KUKA KRL program: MyProgram_223().src

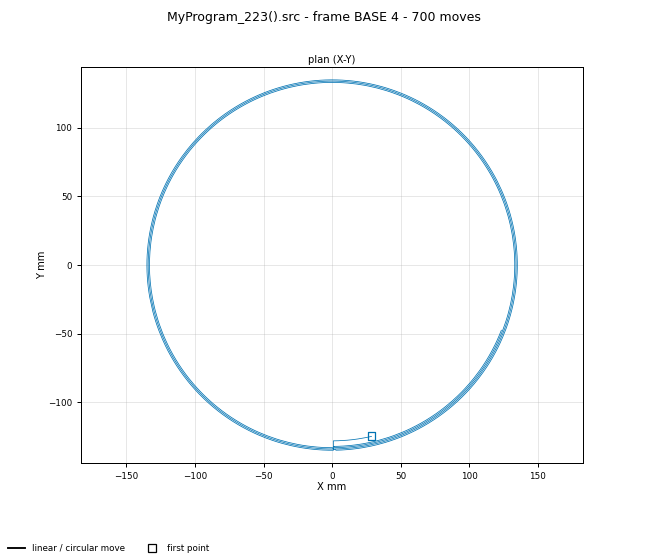
[picture p0: tool path of MyProgram_223().src in frame BASE 4, 700 of 700 moves have a stored position in this frame; points joined in program order, loops and branches not executed]
&ACCESS RVP
&REL 1
&PARAM TEMPLATE = C:\KRC\Roboter\Template\vorgabe
&PARAM EDITMASK = *
DEF MyProgram_223()
; ---- Setting reference (Base) ----
$BASE = BASE_DATA[4]

; --------------------------
; ---- Setting tool (TCP) ----
$TOOL = TOOL_DATA[3]
; --------------------------

$VEL.CP = VEL_APROX_PRINT
Startdeposition()
$VEL.CP = VEL_PRINT
LIN {X 28.7069,Y -124.9653,Z 154,A -77.9995,B 16.837,C -0.17,E1 16.8732,E2 526.8785} C_DIS
LIN {X 25.0095,Y -125.7587,Z 154,A -79.6825,B 16.837,C -0.1689,E1 16.8686,E2 528.562} C_DIS
LIN {X 21.848,Y -126.3473,Z 154,A -81.1205,B 16.837,C -0.1678,E1 16.8647,E2 530.0012} C_DIS
LIN {X 18.7921,Y -126.8373,Z 154,A -82.6165,B 16.837,C -0.1631,E1 16.8605,E2 531.5113} C_DIS
LIN {X 14.8187,Y -127.3616,Z 154,A -84.2756,B 16.837,C -0.1666,E1 16.8559,E2 533.1562} C_DIS
LIN {X 10.9976,Y -127.7479,Z 154,A -86.0056,B 16.837,C -0.1654,E1 16.8511,E2 534.8888} C_DIS
LIN {X 7.8618,Y -127.979,Z 154,A -87.4025,B 16.837,C -0.1651,E1 16.8472,E2 536.2856} C_DIS
LIN {X 4.7214,Y -128.1337,Z 154,A -88.9391,B 16.837,C -0.1603,E1 16.8429,E2 537.8382} C_DIS
LIN {X 0.8945,Y -128.2158,Z 154,A -89.9476,B 16.8368,C -0.1836,E1 16.8403,E2 538.7658} C_DIS
Enddeposition()
LIN {X 0.956,Y -135.0652,Z 155,A -92.2776,B 24.9684,C -1.2991,E1 25.0025,E2 538.84} C_DIS
Startdeposition()
$VEL.CP = VEL_PRINT
LIN {X -2.5758,Y -135.0444,Z 155,A -94.5411,B 24.9704,C -1.2578,E1 24.996,E2 541.2013} C_DIS
LIN {X -6.7331,Y -134.9006,Z 155,A -96.2372,B 24.9702,C -1.2612,E1 24.9912,E2 542.8895} C_DIS
LIN {X -10.9178,Y -134.6272,Z 155,A -98.0533,B 24.9703,C -1.2593,E1 24.9862,E2 544.711} C_DIS
LIN {X -14.6224,Y -134.2747,Z 155,A -99.5996,B 24.9703,C -1.2612,E1 24.9819,E2 546.2538} C_DIS
LIN {X -18.9041,Y -133.7391,Z 155,A -101.4287,B 24.9702,C -1.2616,E1 24.9768,E2 548.0831} C_DIS
LIN {X -22.4797,Y -133.1848,Z 155,A -102.9613,B 24.9702,C -1.2622,E1 24.9726,E2 549.6158} C_DIS
LIN {X -26.677,Y -132.4079,Z 155,A -104.759,B 24.9701,C -1.2636,E1 24.9677,E2 551.4121} C_DIS
LIN {X -30.089,Y -131.6741,Z 155,A -106.2282,B 24.9701,C -1.2649,E1 24.9637,E2 552.8801} C_DIS
LIN {X -33.3739,Y -130.8802,Z 155,A -107.6389,B 24.9699,C -1.2669,E1 24.9599,E2 554.2879} C_DIS
LIN {X -36.516,Y -130.0385,Z 155,A -109.0601,B 24.9699,C -1.2657,E1 24.956,E2 555.7143} C_DIS
LIN {X -39.7548,Y -129.0853,Z 155,A -110.482,B 24.9699,C -1.2672,E1 24.9522,E2 557.1349} C_DIS
LIN {X -43.4103,Y -127.9044,Z 155,A -112.2658,B 24.9702,C -1.2605,E1 24.9474,E2 558.9378} C_DIS
LIN {X -48.0128,Y -126.2483,Z 155,A -114.1681,B 24.9697,C -1.2714,E1 24.9425,E2 560.8182} C_DIS
LIN {X -50.9174,Y -125.104,Z 155,A -115.4973,B 24.9697,C -1.2725,E1 24.9391,E2 562.1477} C_DIS
LIN {X -53.8737,Y -123.8591,Z 155,A -116.8849,B 24.9697,C -1.2726,E1 24.9355,E2 563.5383} C_DIS
LIN {X -57.0265,Y -122.4397,Z 155,A -118.3499,B 24.9696,C -1.2744,E1 24.9318,E2 565.0027} C_DIS
LIN {X -60.55,Y -120.7382,Z 155,A -120.1373,B 24.9698,C -1.2699,E1 24.9273,E2 566.8054} C_DIS
LIN {X -64.3446,Y -118.7594,Z 155,A -121.9404,B 24.9696,C -1.273,E1 24.9228,E2 568.6063} C_DIS
LIN {X -68.1625,Y -116.6098,Z 155,A -123.8138,B 24.9696,C -1.2749,E1 24.9183,E2 570.4805} C_DIS
LIN {X -72.0026,Y -114.2783,Z 155,A -125.7043,B 24.9694,C -1.2787,E1 24.9138,E2 572.3682} C_DIS
LIN {X -75.5548,Y -111.9616,Z 155,A -127.5227,B 24.9693,C -1.2806,E1 24.9096,E2 574.1878} C_DIS
LIN {X -79.2894,Y -109.3484,Z 155,A -129.4475,B 24.9691,C -1.2844,E1 24.9052,E2 576.1102} C_DIS
LIN {X -82.9569,Y -106.5932,Z 155,A -131.4123,B 24.969,C -1.287,E1 24.9008,E2 578.076} C_DIS
LIN {X -86.4643,Y -103.7689,Z 155,A -133.3577,B 24.9689,C -1.2889,E1 24.8966,E2 580.0244} C_DIS
LIN {X -89.8678,Y -100.8354,Z 155,A -135.2713,B 24.9687,C -1.2924,E1 24.8926,E2 581.9372} C_DIS
LIN {X -93.2442,Y -97.7211,Z 155,A -137.1683,B 24.9684,C -1.2991,E1 24.8887,E2 583.826} C_DIS
LIN {X -96.9915,Y -94.0028,Z 155,A -139.3932,B 24.9681,C -1.3047,E1 24.8844,E2 586.047} C_DIS
LIN {X -99.861,Y -90.9491,Z 155,A -141.2062,B 24.9681,C -1.3069,E1 24.8809,E2 587.8626} C_DIS
LIN {X -102.662,Y -87.7755,Z 155,A -142.9452,B 24.9677,C -1.314,E1 24.8778,E2 589.5927} C_DIS
LIN {X -105.1,Y -84.8403,Z 155,A -144.6551,B 24.9677,C -1.3133,E1 24.8747,E2 591.3121} C_DIS
LIN {X -108.2093,Y -80.8373,Z 155,A -146.8037,B 24.9674,C -1.3188,E1 24.8711,E2 593.458} C_DIS
LIN {X -110.7077,Y -77.3807,Z 155,A -148.6369,B 24.9673,C -1.3222,E1 24.8681,E2 595.292} C_DIS
LIN {X -113.1135,Y -73.8196,Z 155,A -150.4801,B 24.9671,C -1.326,E1 24.8653,E2 597.1353} C_DIS
LIN {X -115.3987,Y -70.1936,Z 155,A -152.3394,B 24.9669,C -1.3289,E1 24.8625,E2 598.9974} C_DIS
LIN {X -117.7263,Y -66.2149,Z 155,A -154.2561,B 24.9666,C -1.3362,E1 24.8599,E2 600.9066} C_DIS
LIN {X -119.7417,Y -62.4932,Z 155,A -155.9961,B 24.9662,C -1.344,E1 24.8576,E2 602.6371} C_DIS
LIN {X -121.6486,Y -58.6962,Z 155,A -157.6914,B 24.9656,C -1.3545,E1 24.8555,E2 604.3166} C_DIS
LIN {X -123.7406,Y -54.1479,Z 155,A -159.8366,B 24.9654,C -1.3596,E1 24.853,E2 606.4614} C_DIS
LIN {X -125.3816,Y -50.2287,Z 155,A -161.6964,B 24.9652,C -1.3621,E1 24.851,E2 608.3256} C_DIS
LIN {X -126.4676,Y -47.427,Z 155,A -163.026,B 24.9652,C -1.3633,E1 24.8497,E2 609.66} C_DIS
LIN {X -127.6173,Y -44.2406,Z 155,A -164.4544,B 24.9649,C -1.3681,E1 24.8484,E2 611.085} C_DIS
LIN {X -128.7101,Y -40.953,Z 155,A -165.9753,B 24.9649,C -1.3701,E1 24.8471,E2 612.6098} C_DIS
LIN {X -129.859,Y -37.1578,Z 155,A -167.9428,B 24.9653,C -1.3613,E1 24.8455,E2 614.6097} C_DIS
LIN {X -130.7137,Y -34.0292,Z 155,A -169.0198,B 24.9643,C -1.3802,E1 24.8448,E2 615.6478} C_DIS
LIN {X -133.0003,Y -23.5463,Z 155,A -173.6124,B 24.9637,C -1.3927,E1 24.8421,E2 620.2378} C_DIS
LIN {X -133.6072,Y -19.827,Z 155,A -175.3609,B 24.9637,C -1.3905,E1 24.8413,E2 622.002} C_DIS
LIN {X -134.12,Y -15.9779,Z 155,A -176.8994,B 24.9632,C -1.4012,E1 24.8408,E2 623.5241} C_DIS
LIN {X -134.4898,Y -12.4963,Z 155,A -178.3737,B 24.9629,C -1.4066,E1 24.8404,E2 624.9944} C_DIS
LIN {X -134.7979,Y -8.5494,Z 155,A 179.9081,B 24.9627,C -1.4102,E1 24.84,E2 626.7143} C_DIS
LIN {X -134.9759,Y -5.0083,Z 155,A 178.3069,B 24.9627,C -1.4104,E1 24.8399,E2 628.3247} C_DIS
LIN {X -135.0684,Y -0.5524,Z 155,A 176.4249,B 24.9624,C -1.4171,E1 24.8398,E2 630.2022} C_DIS
LIN {X -135.0185,Y 3.6788,Z 155,A 174.6963,B 24.9619,C -1.4263,E1 24.8398,E2 631.9192} C_DIS
LIN {X -134.8642,Y 7.4574,Z 155,A 172.9572,B 24.9619,C -1.425,E1 24.8401,E2 633.6718} C_DIS
LIN {X -134.5797,Y 11.4806,Z 155,A 171.3594,B 24.9614,C -1.4362,E1 24.8405,E2 635.2525} C_DIS
LIN {X -134.165,Y 15.6009,Z 155,A 169.5519,B 24.9612,C -1.4395,E1 24.841,E2 637.0629} C_DIS
LIN {X -133.7051,Y 19.1415,Z 155,A 168.0667,B 24.9608,C -1.446,E1 24.8416,E2 638.5416} C_DIS
LIN {X -133.0954,Y 23.0147,Z 155,A 166.2283,B 24.961,C -1.4429,E1 24.8424,E2 640.3984} C_DIS
LIN {X -132.3123,Y 27.1467,Z 155,A 164.5508,B 24.9604,C -1.454,E1 24.8433,E2 642.0594} C_DIS
LIN {X -131.1469,Y 32.3169,Z 155,A 162.3649,B 24.9598,C -1.4643,E1 24.8447,E2 644.2333} C_DIS
LIN {X -130.3875,Y 35.2526,Z 155,A 160.9043,B 24.9601,C -1.46,E1 24.8457,E2 645.7127} C_DIS
LIN {X -129.1991,Y 39.3831,Z 155,A 158.5311,B 24.9612,C -1.4393,E1 24.8477,E2 648.1491} C_DIS
LIN {X -127.5792,Y 44.3504,Z 155,A 156.9773,B 24.959,C -1.4785,E1 24.849,E2 649.6183} C_DIS
LIN {X -126.4051,Y 47.5939,Z 155,A 155.4977,B 24.9588,C -1.4823,E1 24.8504,E2 651.0971} C_DIS
LIN {X -125.2195,Y 50.6307,Z 155,A 154.1008,B 24.9586,C -1.486,E1 24.8519,E2 652.493} C_DIS
LIN {X -123.8761,Y 53.8345,Z 155,A 152.6264,B 24.9584,C -1.4906,E1 24.8535,E2 653.9647} C_DIS
LIN {X -122.507,Y 56.8809,Z 155,A 151.1945,B 24.9582,C -1.4942,E1 24.8552,E2 655.3957} C_DIS
LIN {X -120.9936,Y 60.0334,Z 155,A 149.6811,B 24.958,C -1.4973,E1 24.857,E2 656.9101} C_DIS
LIN {X -119.2067,Y 63.5116,Z 155,A 147.8717,B 24.9581,C -1.4949,E1 24.8594,E2 658.7348} C_DIS
LIN {X -116.8772,Y 67.7024,Z 155,A 145.8996,B 24.9576,C -1.504,E1 24.8621,E2 660.6955} C_DIS
LIN {X -114.4989,Y 71.6521,Z 155,A 143.9181,B 24.9574,C -1.5084,E1 24.865,E2 662.6766} C_DIS
LIN {X -112.0741,Y 75.3886,Z 155,A 141.9947,B 24.9572,C -1.5122,E1 24.8679,E2 664.6007} C_DIS
LIN {X -109.5159,Y 79.0583,Z 155,A 140.1208,B 24.9568,C -1.5187,E1 24.8709,E2 666.4682} C_DIS
LIN {X -105.4703,Y 84.3802,Z 155,A 137.3252,B 24.9562,C -1.5284,E1 24.8757,E2 669.254} C_DIS
LIN {X -101.5038,Y 89.1125,Z 155,A 134.5151,B 24.9564,C -1.526,E1 24.8808,E2 672.0828} C_DIS
LIN {X -97.5119,Y 93.4631,Z 155,A 132.2969,B 24.9552,C -1.5465,E1 24.885,E2 674.2618} C_DIS
LIN {X -95.259,Y 95.7581,Z 155,A 130.7619,B 24.9555,C -1.5415,E1 24.888,E2 675.8154} C_DIS
LIN {X -92.1865,Y 98.7196,Z 155,A 128.877,B 24.9555,C -1.5421,E1 24.8919,E2 677.7064} C_DIS
LIN {X -88.0432,Y 102.4319,Z 155,A 126.8279,B 24.9542,C -1.5631,E1 24.8961,E2 679.7137} C_DIS
LIN {X -85.7976,Y 104.3208,Z 155,A 125.2543,B 24.955,C -1.5495,E1 24.8995,E2 681.3255} C_DIS
LIN {X -82.2968,Y 107.1038,Z 155,A 122.8357,B 24.9563,C -1.5279,E1 24.905,E2 683.8044} C_DIS
LIN {X -78.1726,Y 110.1502,Z 155,A 121.4737,B 24.9537,C -1.5728,E1 24.9079,E2 685.0644} C_DIS
LIN {X -73.9894,Y 113.0026,Z 155,A 119.0337,B 24.9543,C -1.5625,E1 24.9136,E2 687.537} C_DIS
LIN {X -70.0577,Y 115.4809,Z 155,A 117.0561,B 24.9541,C -1.566,E1 24.9183,E2 689.5126} C_DIS
LIN {X -66.2162,Y 117.7256,Z 155,A 115.1687,B 24.9539,C -1.5694,E1 24.9228,E2 691.3975} C_DIS
LIN {X -62.6191,Y 119.6756,Z 155,A 113.5082,B 24.9534,C -1.5762,E1 24.9269,E2 693.0464} C_DIS
LIN {X -59.6022,Y 121.2063,Z 155,A 112.069,B 24.9534,C -1.5784,E1 24.9305,E2 694.4842} C_DIS
LIN {X -56.3004,Y 122.7755,Z 155,A 110.5474,B 24.9531,C -1.5823,E1 24.9343,E2 696.0005} C_DIS
LIN {X -53.2438,Y 124.1315,Z 155,A 109.0926,B 24.9531,C -1.5826,E1 24.938,E2 697.458} C_DIS
LIN {X -49.3123,Y 125.7451,Z 155,A 107.2368,B 24.9531,C -1.5825,E1 24.9429,E2 699.3181} C_DIS
LIN {X -45.9259,Y 127.0206,Z 155,A 105.74,B 24.9528,C -1.5864,E1 24.9468,E2 700.8085} C_DIS
LIN {X -42.4672,Y 128.2185,Z 155,A 104.2256,B 24.9526,C -1.5903,E1 24.9507,E2 702.3166} C_DIS
LIN {X -39.232,Y 129.2453,Z 155,A 102.7595,B 24.9526,C -1.5907,E1 24.9547,E2 703.7844} C_DIS
LIN {X -35.3424,Y 130.3635,Z 155,A 100.9587,B 24.9527,C -1.5882,E1 24.9595,E2 705.5939} C_DIS
LIN {X -31.7612,Y 131.2809,Z 155,A 99.444,B 24.9525,C -1.5925,E1 24.9636,E2 707.1005} C_DIS
LIN {X -28.1853,Y 132.0951,Z 155,A 97.9093,B 24.9523,C -1.595,E1 24.9678,E2 708.6312} C_DIS
LIN {X -24.1975,Y 132.8838,Z 155,A 96.1246,B 24.9524,C -1.5933,E1 24.9727,E2 710.4219} C_DIS
LIN {X -20.4636,Y 133.5093,Z 155,A 94.597,B 24.9521,C -1.5985,E1 24.9769,E2 711.9386} C_DIS
LIN {X -17.178,Y 133.9721,Z 155,A 93.0679,B 24.9524,C -1.5931,E1 24.9811,E2 713.4815} C_DIS
LIN {X -12.8968,Y 134.4513,Z 155,A 91.3198,B 24.9521,C -1.5982,E1 24.986,E2 715.2187} C_DIS
LIN {X -8.8291,Y 134.7806,Z 155,A 89.5073,B 24.9523,C -1.5948,E1 24.991,E2 717.04} C_DIS
LIN {X -4.9442,Y 134.9784,Z 155,A 87.8488,B 24.9523,C -1.5948,E1 24.9957,E2 718.6986} C_DIS
LIN {X -0.6766,Y 135.0669,Z 155,A 86.1042,B 24.9521,C -1.5988,E1 25.0005,E2 720.4341} C_DIS
LIN {X 3.559,Y 135.0218,Z 155,A 84.3207,B 24.9521,C -1.5997,E1 25.0055,E2 722.2151} C_DIS
LIN {X 7.3645,Y 134.8688,Z 155,A 82.605,B 24.9524,C -1.5945,E1 25.0103,E2 723.9426} C_DIS
LIN {X 11.3614,Y 134.5898,Z 155,A 81.0168,B 24.952,C -1.6003,E1 25.0147,E2 725.5163} C_DIS
LIN {X 15.2359,Y 134.2085,Z 155,A 79.2316,B 24.9525,C -1.593,E1 25.0197,E2 727.3176} C_DIS
LIN {X 19.1015,Y 133.7109,Z 155,A 77.7249,B 24.952,C -1.6003,E1 25.0238,E2 728.8057} C_DIS
LIN {X 22.5739,Y 133.169,Z 155,A 76.1081,B 24.9524,C -1.5932,E1 25.0283,E2 730.4378} C_DIS
LIN {X 26.8961,Y 132.3633,Z 155,A 74.3688,B 24.9521,C -1.599,E1 25.033,E2 732.1613} C_DIS
LIN {X 30.2156,Y 131.6452,Z 155,A 72.9373,B 24.9521,C -1.5987,E1 25.0369,E2 733.5915} C_DIS
LIN {X 33.4163,Y 130.8694,Z 155,A 71.524,B 24.9522,C -1.597,E1 25.0408,E2 735.0067} C_DIS
LIN {X 36.6251,Y 130.008,Z 155,A 70.1141,B 24.9522,C -1.596,E1 25.0446,E2 736.4168} C_DIS
LIN {X 40.4048,Y 128.8852,Z 155,A 68.3482,B 24.9526,C -1.5897,E1 25.0493,E2 738.1943} C_DIS
LIN {X 45.0769,Y 127.3266,Z 155,A 66.3968,B 24.9523,C -1.5952,E1 25.0544,E2 740.1289} C_DIS
LIN {X 47.6833,Y 126.3716,Z 155,A 65.2107,B 24.9524,C -1.5936,E1 25.0575,E2 741.3163} C_DIS
LIN {X 50.746,Y 125.1731,Z 155,A 63.7899,B 24.9526,C -1.5908,E1 25.0612,E2 742.7406} C_DIS
LIN {X 53.8201,Y 123.8823,Z 155,A 62.393,B 24.9526,C -1.5902,E1 25.0648,E2 744.1356} C_DIS
LIN {X 56.9496,Y 122.4753,Z 155,A 60.9484,B 24.9526,C -1.589,E1 25.0685,E2 745.5794} C_DIS
LIN {X 60.0444,Y 120.9882,Z 155,A 59.4823,B 24.9528,C -1.5866,E1 25.0722,E2 747.0472} C_DIS
LIN {X 63.2089,Y 119.3659,Z 155,A 57.9622,B 24.953,C -1.584,E1 25.0759,E2 748.5694} C_DIS
LIN {X 66.9392,Y 117.316,Z 155,A 56.0485,B 24.9535,C -1.5755,E1 25.0806,E2 750.4973} C_DIS
LIN {X 70.8345,Y 115.0062,Z 155,A 54.2606,B 24.9532,C -1.5797,E1 25.0849,E2 752.2697} C_DIS
LIN {X 74.1026,Y 112.928,Z 155,A 52.5215,B 24.9537,C -1.5719,E1 25.089,E2 754.0218} C_DIS
LIN {X 77.8951,Y 110.346,Z 155,A 50.6151,B 24.9537,C -1.5707,E1 25.0933,E2 755.9245} C_DIS
LIN {X 81.529,Y 107.6892,Z 155,A 48.716,B 24.9539,C -1.5678,E1 25.0976,E2 757.8237} C_DIS
LIN {X 85.0807,Y 104.9061,Z 155,A 46.8107,B 24.9541,C -1.5646,E1 25.1018,E2 759.7293} C_DIS
LIN {X 88.2784,Y 102.2293,Z 155,A 45.0412,B 24.9543,C -1.561,E1 25.1055,E2 761.5003} C_DIS
LIN {X 91.5574,Y 99.3034,Z 155,A 43.1894,B 24.9545,C -1.5579,E1 25.1094,E2 763.3521} C_DIS
LIN {X 94.7667,Y 96.2456,Z 155,A 41.2984,B 24.9548,C -1.5532,E1 25.1132,E2 765.2462} C_DIS
LIN {X 97.9192,Y 93.0369,Z 155,A 39.433,B 24.9549,C -1.5513,E1 25.1168,E2 767.1082} C_DIS
LIN {X 100.8417,Y 89.8607,Z 155,A 37.6085,B 24.9551,C -1.5474,E1 25.1202,E2 768.9338} C_DIS
LIN {X 103.6576,Y 86.5972,Z 155,A 35.7454,B 24.9555,C -1.5411,E1 25.1236,E2 770.8032} C_DIS
LIN {X 106.466,Y 83.1206,Z 155,A 33.8428,B 24.9558,C -1.536,E1 25.1269,E2 772.7088} C_DIS
LIN {X 109.1862,Y 79.5132,Z 155,A 31.9399,B 24.956,C -1.5319,E1 25.1301,E2 774.6123} C_DIS
LIN {X 111.7145,Y 75.9199,Z 155,A 30.089,B 24.9563,C -1.5278,E1 25.133,E2 776.4639} C_DIS
LIN {X 114.2202,Y 72.0947,Z 155,A 28.1796,B 24.9565,C -1.5243,E1 25.1359,E2 778.372} C_DIS
LIN {X 116.5986,Y 68.1817,Z 155,A 26.2431,B 24.9568,C -1.5193,E1 25.1387,E2 780.3104} C_DIS
LIN {X 118.7941,Y 64.2807,Z 155,A 24.3469,B 24.9571,C -1.5141,E1 25.1412,E2 782.2089} C_DIS
LIN {X 120.525,Y 60.9688,Z 155,A 22.9027,B 24.9569,C -1.5174,E1 25.1431,E2 783.6375} C_DIS
LIN {X 121.9558,Y 58.0532,Z 155,A 21.5126,B 24.9571,C -1.5128,E1 25.1447,E2 785.0312} C_DIS
LIN {X 123.3484,Y 55.0323,Z 155,A 20.1045,B 24.9574,C -1.5088,E1 25.1464,E2 786.4411} C_DIS
LIN {X 124.7016,Y 51.8933,Z 155,A 18.6636,B 24.9576,C -1.505,E1 25.1479,E2 787.8829} C_DIS
LIN {X 125.9888,Y 48.6856,Z 155,A 17.2055,B 24.9578,C -1.501,E1 25.1494,E2 789.3423} C_DIS
LIN {X 127.4202,Y 44.809,Z 155,A 15.3011,B 24.9586,C -1.4872,E1 25.1513,E2 791.2685} C_DIS
LIN {X 128.9009,Y 40.3554,Z 155,A 13.139,B 24.9594,C -1.4715,E1 25.1531,E2 793.4554} C_DIS
LIN {X 129.9101,Y 36.9751,Z 155,A 12.0923,B 24.9583,C -1.492,E1 25.1539,E2 794.448} C_DIS
LIN {X 130.9776,Y 32.99,Z 155,A 10.2421,B 24.9589,C -1.4808,E1 25.1552,E2 796.3137} C_DIS
LIN {X 131.967,Y 28.7787,Z 155,A 8.4174,B 24.9592,C -1.4756,E1 25.1564,E2 798.1402} C_DIS
LIN {X 132.6716,Y 25.3314,Z 155,A 6.9657,B 24.9593,C -1.4731,E1 25.1571,E2 799.5894} C_DIS
LIN {X 133.2979,Y 21.8018,Z 155,A 5.4671,B 24.9596,C -1.4694,E1 25.1578,E2 801.0878} C_DIS
LIN {X 133.865,Y 17.9954,Z 155,A 3.7685,B 24.96,C -1.4604,E1 25.1585,E2 802.7978} C_DIS
LIN {X 134.3238,Y 14.1661,Z 155,A 2.1058,B 24.9604,C -1.4535,E1 25.159,E2 804.4667} C_DIS
LIN {X 134.7085,Y 9.854,Z 155,A 0.3864,B 24.9604,C -1.4541,E1 25.1594,E2 806.1746} C_DIS
LIN {X 134.9165,Y 6.416,Z 155,A -1.1834,B 24.961,C -1.4431,E1 25.1597,E2 807.7609} C_DIS
LIN {X 135.0499,Y 2.2472,Z 155,A -2.8475,B 24.961,C -1.4431,E1 25.1597,E2 809.415} C_DIS
LIN {X 135.0526,Y -2.0829,Z 155,A -4.687,B 24.9613,C -1.4369,E1 25.1597,E2 811.2582} C_DIS
LIN {X 134.9392,Y -5.9477,Z 155,A -6.3919,B 24.9618,C -1.4278,E1 25.1596,E2 812.9744} C_DIS
LIN {X 134.7122,Y -9.8033,Z 155,A -7.8928,B 24.9617,C -1.4301,E1 25.1593,E2 814.461} C_DIS
LIN {X 134.4232,Y -13.1893,Z 155,A -9.4289,B 24.9622,C -1.42,E1 25.1589,E2 816.0118} C_DIS
LIN {X 133.938,Y -17.4382,Z 155,A -11.1522,B 24.9622,C -1.4191,E1 25.1583,E2 817.7271} C_DIS
LIN {X 133.4162,Y -21.0649,Z 155,A -12.7866,B 24.9628,C -1.4094,E1 25.1576,E2 819.3746} C_DIS
LIN {X 132.6927,Y -25.2211,Z 155,A -14.4859,B 24.9628,C -1.4086,E1 25.1568,E2 821.066} C_DIS
LIN {X 131.9741,Y -28.7461,Z 155,A -15.967,B 24.963,C -1.4061,E1 25.1559,E2 822.5443} C_DIS
LIN {X 131.1265,Y -32.4017,Z 155,A -17.6861,B 24.9636,C -1.3937,E1 25.1548,E2 824.2827} C_DIS
LIN {X 130.1075,Y -36.2695,Z 155,A -19.2728,B 24.9636,C -1.3944,E1 25.1537,E2 825.8587} C_DIS
LIN {X 129.1637,Y -39.4988,Z 155,A -20.6741,B 24.9637,C -1.3912,E1 25.1525,E2 827.2594} C_DIS
LIN {X 128.1047,Y -42.8088,Z 155,A -22.1386,B 24.964,C -1.387,E1 25.1513,E2 828.7256} C_DIS
LIN {X 126.7849,Y -46.5796,Z 155,A -24.1151,B 24.9651,C -1.3658,E1 25.1494,E2 830.741} C_DIS
LIN {X 125.5935,Y -49.7023,Z 155,A -25.2102,B 24.9644,C -1.3794,E1 25.1483,E2 831.798} C_DIS
LIN {X 124.5325,Y -52.2983,Z 155,A -26.5775,B 24.9651,C -1.3657,E1 25.1468,E2 833.1901} C_DIS
LIN {X 122.5054,Y -56.8843,Z 155,A -28.5105,B 24.9648,C -1.3699,E1 25.1446,E2 835.1025} C_DIS
LIN {X 121.0419,Y -59.9355,Z 155,A -29.9491,B 24.9651,C -1.3653,E1 25.1428,E2 836.5443} C_DIS
LIN {X 119.2537,Y -63.4225,Z 155,A -31.6529,B 24.9655,C -1.3579,E1 25.1406,E2 838.2565} C_DIS
LIN {X 117.1158,Y -67.29,Z 155,A -33.5556,B 24.9658,C -1.3507,E1 25.138,E2 840.1664} C_DIS
LIN {X 114.8507,Y -71.0866,Z 155,A -35.3212,B 24.9658,C -1.3513,E1 25.1355,E2 841.9215} C_DIS
LIN {X 112.8245,Y -74.2598,Z 155,A -36.9709,B 24.9662,C -1.3437,E1 25.1329,E2 843.5808} C_DIS
LIN {X 110.302,Y -77.9575,Z 155,A -38.8612,B 24.9664,C -1.3388,E1 25.1299,E2 845.4736} C_DIS
LIN {X 106.7912,Y -82.7014,Z 155,A -40.9817,B 24.9657,C -1.3532,E1 25.1265,E2 847.5498} C_DIS
LIN {X 103.6981,Y -86.5489,Z 155,A -43.4463,B 24.967,C -1.3268,E1 25.122,E2 850.0653} C_DIS
LIN {X 100.9103,Y -89.784,Z 155,A -45.2755,B 24.9673,C -1.321,E1 25.1187,E2 851.9} C_DIS
LIN {X 97.8876,Y -93.0699,Z 155,A -47.1747,B 24.9676,C -1.3158,E1 25.115,E2 853.803} C_DIS
LIN {X 94.7246,Y -96.287,Z 155,A -49.061,B 24.9677,C -1.3125,E1 25.1113,E2 855.6891} C_DIS
LIN {X 91.4798,Y -99.3747,Z 155,A -50.9353,B 24.9679,C -1.3093,E1 25.1075,E2 857.5632} C_DIS
LIN {X 88.0317,Y -102.4419,Z 155,A -52.8541,B 24.968,C -1.3069,E1 25.1035,E2 859.4802} C_DIS
LIN {X 84.8065,Y -105.1273,Z 155,A -54.6442,B 24.9682,C -1.3023,E1 25.0996,E2 861.2744} C_DIS
LIN {X 81.2739,Y -107.8817,Z 155,A -56.5402,B 24.9684,C -1.2983,E1 25.0954,E2 863.1728} C_DIS
LIN {X 77.5783,Y -110.5695,Z 155,A -58.4279,B 24.9684,C -1.297,E1 25.0911,E2 865.057} C_DIS
LIN {X 74.1604,Y -112.8899,Z 155,A -60.1684,B 24.9686,C -1.2941,E1 25.0871,E2 866.7986} C_DIS
LIN {X 70.4829,Y -115.2219,Z 155,A -62.0101,B 24.9688,C -1.2908,E1 25.0827,E2 868.6422} C_DIS
LIN {X 66.0835,Y -117.8001,Z 155,A -64.2026,B 24.9691,C -1.2852,E1 25.0774,E2 870.8414} C_DIS
LIN {X 62.536,Y -119.7192,Z 155,A -65.8308,B 24.969,C -1.2867,E1 25.0734,E2 872.4613} C_DIS
LIN {X 59.4854,Y -121.2639,Z 155,A -67.2607,B 24.969,C -1.2854,E1 25.0698,E2 873.8904} C_DIS
LIN {X 56.4805,Y -122.6922,Z 155,A -68.6813,B 24.9692,C -1.2826,E1 25.0662,E2 875.3141} C_DIS
LIN {X 53.3322,Y -124.0932,Z 155,A -70.1201,B 24.9692,C -1.2816,E1 25.0625,E2 876.7517} C_DIS
LIN {X 50.2793,Y -125.3612,Z 155,A -71.5253,B 24.9693,C -1.2794,E1 25.0589,E2 878.159} C_DIS
LIN {X 47.0377,Y -126.6135,Z 155,A -73.2727,B 24.9701,C -1.2625,E1 25.0542,E2 879.9426} C_DIS
LIN {X 42.5301,Y -128.1976,Z 155,A -75.4538,B 24.9707,C -1.2515,E1 25.0484,E2 882.1453} C_DIS
LIN {X 38.6214,Y -129.4306,Z 155,A -76.701,B 24.9695,C -1.276,E1 25.0452,E2 883.3323} C_DIS
LIN {X 32.826,Y -131.0193,Z 155,A -79.4265,B 24.9701,C -1.2637,E1 25.0378,E2 886.0827} C_DIS
LIN {X 28.6739,Y -131.9897,Z 155,A -81.1094,B 24.9699,C -1.2688,E1 25.0333,E2 887.7514} C_DIS
LIN {X 25.3059,Y -132.6765,Z 155,A -82.5595,B 24.9699,C -1.2679,E1 25.0293,E2 889.2017} C_DIS
LIN {X 22.1238,Y -133.2441,Z 155,A -83.9504,B 24.9699,C -1.2658,E1 25.0255,E2 890.5961} C_DIS
LIN {X 18.3516,Y -133.818,Z 155,A -85.681,B 24.9703,C -1.2586,E1 25.0206,E2 892.3423} C_DIS
LIN {X 14.4787,Y -134.2902,Z 155,A -87.2046,B 24.97,C -1.2647,E1 25.0165,E2 893.8504} C_DIS
LIN {X 11.0079,Y -134.6196,Z 155,A -88.7435,B 24.9702,C -1.2607,E1 25.0122,E2 895.3979} C_DIS
LIN {X 6.8304,Y -134.8957,Z 155,A -90.4623,B 24.9702,C -1.263,E1 25.0074,E2 897.1105} C_DIS
LIN {X 3.0442,Y -135.0361,Z 155,A -92.1772,B 24.9704,C -1.2567,E1 25.0025,E2 898.84} C_DIS
LIN {X 3.0442,Y -135.0361,Z 155,A -92.1772,B 24.9704,C -1.2567,E1 25.0025,E2 898.84} C_DIS
Enddeposition()
LIN {X 0.9544,Y -134.1287,Z 155,A -92.5293,B 23.7995,C -1.0605,E1 23.8224,E2 899.5208} C_DIS
Startdeposition()
$VEL.CP = VEL_PRINT
LIN {X 3.395,Y -134.0907,Z 155,A -90.8525,B 23.7982,C -1.0929,E1 23.8273,E2 897.7641} C_DIS
LIN {X 6.9399,Y -133.9537,Z 155,A -89.3571,B 23.7982,C -1.0925,E1 23.8315,E2 896.2703} C_DIS
LIN {X 11.1296,Y -133.6707,Z 155,A -87.566,B 23.7982,C -1.0932,E1 23.8365,E2 894.4784} C_DIS
LIN {X 14.863,Y -133.3081,Z 155,A -85.8806,B 23.7979,C -1.0983,E1 23.8412,E2 892.7815} C_DIS
LIN {X 18.8851,Y -132.797,Z 155,A -84.2368,B 23.7981,C -1.0949,E1 23.8457,E2 891.1475} C_DIS
LIN {X 22.8343,Y -132.1774,Z 155,A -82.4743,B 23.7979,C -1.099,E1 23.8506,E2 889.3768} C_DIS
LIN {X 26.6564,Y -131.4576,Z 155,A -80.8841,B 23.7979,C -1.0968,E1 23.8549,E2 887.794} C_DIS
LIN {X 29.9513,Y -130.7463,Z 155,A -79.4604,B 23.7979,C -1.0973,E1 23.8588,E2 886.3711} C_DIS
LIN {X 32.6881,Y -130.0893,Z 155,A -77.8581,B 23.797,C -1.1193,E1 23.8633,E2 884.7169} C_DIS
LIN {X 36.3324,Y -129.1187,Z 155,A -76.6081,B 23.7978,C -1.1023,E1 23.8665,E2 883.5112} C_DIS
LIN {X 40.3535,Y -127.9197,Z 155,A -74.8173,B 23.7977,C -1.1043,E1 23.8713,E2 881.7189} C_DIS
LIN {X 43.8741,Y -126.7544,Z 155,A -73.4044,B 23.798,C -1.0974,E1 23.875,E2 880.3258} C_DIS
LIN {X 47.4196,Y -125.4717,Z 155,A -71.5554,B 23.7973,C -1.1119,E1 23.8799,E2 878.445} C_DIS
LIN {X 51.4349,Y -123.8795,Z 155,A -69.8167,B 23.7975,C -1.109,E1 23.8844,E2 876.7176} C_DIS
LIN {X 54.5618,Y -122.5343,Z 155,A -68.4065,B 23.7975,C -1.109,E1 23.888,E2 875.3113} C_DIS
LIN {X 57.586,Y -121.1425,Z 155,A -66.9848,B 23.7974,C -1.1112,E1 23.8916,E2 873.8879} C_DIS
LIN {X 60.5245,Y -119.7017,Z 155,A -65.5715,B 23.7972,C -1.1143,E1 23.8951,E2 872.4709} C_DIS
LIN {X 63.9244,Y -117.9233,Z 155,A -63.807,B 23.7968,C -1.1237,E1 23.8995,E2 870.6884} C_DIS
LIN {X 66.7238,Y -116.3621,Z 155,A -62.3913,B 23.7966,C -1.1287,E1 23.903,E2 869.265} C_DIS
LIN {X 70.6969,Y -113.9917,Z 155,A -60.4519,B 23.7966,C -1.1305,E1 23.9076,E2 867.3276} C_DIS
LIN {X 74.8193,Y -111.3299,Z 155,A -58.4964,B 23.7966,C -1.1272,E1 23.9121,E2 865.3871} C_DIS
LIN {X 78.2609,Y -108.9377,Z 155,A -56.6432,B 23.7963,C -1.1342,E1 23.9164,E2 863.5233} C_DIS
LIN {X 81.8233,Y -106.2884,Z 155,A -54.721,B 23.7961,C -1.1397,E1 23.9207,E2 861.5949} C_DIS
LIN {X 85.3222,Y -103.5003,Z 155,A -52.8295,B 23.7959,C -1.1429,E1 23.9248,E2 859.7031} C_DIS
LIN {X 88.79,Y -100.5408,Z 155,A -50.9396,B 23.7959,C -1.1444,E1 23.9287,E2 857.8174} C_DIS
LIN {X 91.9954,Y -97.6164,Z 155,A -49.0836,B 23.7957,C -1.1489,E1 23.9325,E2 855.9581} C_DIS
LIN {X 95.1832,Y -94.5107,Z 155,A -47.1896,B 23.7955,C -1.1532,E1 23.9363,E2 854.0619} C_DIS
LIN {X 98.3864,Y -91.172,Z 155,A -45.2073,B 23.7952,C -1.1585,E1 23.9401,E2 852.0757} C_DIS
LIN {X 101.3821,Y -87.829,Z 155,A -43.2718,B 23.795,C -1.1645,E1 23.9437,E2 850.1347} C_DIS
LIN {X 104.2077,Y -84.4569,Z 155,A -41.498,B 23.795,C -1.1639,E1 23.9468,E2 848.371} C_DIS
LIN {X 106.4575,Y -81.6023,Z 155,A -39.6621,B 23.7941,C -1.1833,E1 23.95,E2 846.4963} C_DIS
LIN {X 108.5287,Y -78.8267,Z 155,A -38.0967,B 23.7937,C -1.1921,E1 23.9526,E2 844.9174} C_DIS
LIN {X 110.8362,Y -75.5488,Z 155,A -36.8363,B 23.7946,C -1.1726,E1 23.9545,E2 843.7116} C_DIS
LIN {X 112.2454,Y -73.4384,Z 155,A -35.5807,B 23.794,C -1.1849,E1 23.9565,E2 842.4323} C_DIS
LIN {X 114.7605,Y -69.4416,Z 155,A -33.655,B 23.794,C -1.1858,E1 23.9593,E2 840.5145} C_DIS
LIN {X 117.0313,Y -65.5426,Z 155,A -31.7434,B 23.7937,C -1.1906,E1 23.9619,E2 838.6015} C_DIS
LIN {X 119.1959,Y -61.5181,Z 155,A -29.8111,B 23.7935,C -1.1954,E1 23.9644,E2 836.6682} C_DIS
LIN {X 120.9291,Y -58.0326,Z 155,A -28.2848,B 23.7936,C -1.1932,E1 23.9663,E2 835.1561} C_DIS
LIN {X 122.6028,Y -54.4087,Z 155,A -26.4955,B 23.7932,C -1.2029,E1 23.9684,E2 833.353} C_DIS
LIN {X 124.5266,Y -49.8482,Z 155,A -24.4223,B 23.793,C -1.2073,E1 23.9706,E2 831.2811} C_DIS
LIN {X 126.0517,Y -45.8554,Z 155,A -22.5975,B 23.7927,C -1.213,E1 23.9724,E2 829.453} C_DIS
LIN {X 127.2292,Y -42.4778,Z 155,A -21.0991,B 23.7925,C -1.2162,E1 23.9737,E2 827.9556} C_DIS
LIN {X 128.3188,Y -39.0635,Z 155,A -19.5914,B 23.7923,C -1.2198,E1 23.975,E2 826.4479} C_DIS
LIN {X 129.4098,Y -35.2889,Z 155,A -17.8347,B 23.7919,C -1.2294,E1 23.9763,E2 824.6783} C_DIS
LIN {X 130.3607,Y -31.5874,Z 155,A -16.2636,B 23.7918,C -1.2314,E1 23.9774,E2 823.1119} C_DIS
LIN {X 131.2165,Y -27.8231,Z 155,A -14.5442,B 23.7913,C -1.2406,E1 23.9784,E2 821.3805} C_DIS
LIN {X 132.0102,Y -23.7698,Z 155,A -12.9452,B 23.7915,C -1.2374,E1 23.9792,E2 819.7991} C_DIS
LIN {X 132.5567,Y -20.5035,Z 155,A -11.4869,B 23.7911,C -1.2444,E1 23.9799,E2 818.3328} C_DIS
LIN {X 133.1304,Y -16.3782,Z 155,A -9.6709,B 23.7908,C -1.2522,E1 23.9805,E2 816.5088} C_DIS
LIN {X 133.5341,Y -12.6635,Z 155,A -8.1168,B 23.7906,C -1.2551,E1 23.981,E2 814.9571} C_DIS
LIN {X 133.8695,Y -8.4079,Z 155,A -6.3509,B 23.7905,C -1.258,E1 23.9813,E2 813.1952} C_DIS
LIN {X 134.0451,Y -4.8751,Z 155,A -4.7337,B 23.7899,C -1.2687,E1 23.9815,E2 811.5619} C_DIS
LIN {X 134.1332,Y -0.5274,Z 155,A -2.9605,B 23.7899,C -1.2702,E1 23.9815,E2 809.796} C_DIS
LIN {X 134.0852,Y 3.5942,Z 155,A -1.1973,B 23.7896,C -1.2761,E1 23.9815,E2 808.0293} C_DIS
LIN {X 133.9007,Y 7.9025,Z 155,A 0.6341,B 23.7893,C -1.2816,E1 23.9812,E2 806.1961} C_DIS
LIN {X 133.603,Y 11.9318,Z 155,A 2.3926,B 23.7889,C -1.2889,E1 23.9808,E2 804.4304} C_DIS
LIN {X 133.2043,Y 15.7587,Z 155,A 3.9823,B 23.7888,C -1.2913,E1 23.9803,E2 802.8447} C_DIS
LIN {X 132.613,Y 20.1403,Z 155,A 5.8521,B 23.7885,C -1.2964,E1 23.9796,E2 800.9741} C_DIS
LIN {X 132.0374,Y 23.6175,Z 155,A 7.312,B 23.7885,C -1.2987,E1 23.9789,E2 799.5174} C_DIS
LIN {X 131.2882,Y 27.4891,Z 155,A 9.0575,B 23.788,C -1.3073,E1 23.9779,E2 797.7615} C_DIS
LIN {X 130.4238,Y 31.3256,Z 155,A 10.6441,B 23.788,C -1.3076,E1 23.9769,E2 796.1839} C_DIS
LIN {X 129.5989,Y 34.5798,Z 155,A 12.0494,B 23.7878,C -1.3106,E1 23.9759,E2 794.7799} C_DIS
LIN {X 127.9942,Y 40.1203,Z 155,A 14.4913,B 23.7875,C -1.3169,E1 23.974,E2 792.337} C_DIS
LIN {X 126.8167,Y 43.6945,Z 155,A 16.0998,B 23.7872,C -1.3219,E1 23.9725,E2 790.7259} C_DIS
LIN {X 125.7058,Y 46.7945,Z 155,A 17.498,B 23.787,C -1.3257,E1 23.9712,E2 789.3266} C_DIS
LIN {X 124.5061,Y 49.899,Z 155,A 18.8937,B 23.7869,C -1.3285,E1 23.9698,E2 787.9321} C_DIS
LIN {X 123.218,Y 52.9998,Z 155,A 20.3538,B 23.7866,C -1.3341,E1 23.9682,E2 786.4667} C_DIS
LIN {X 121.8233,Y 56.1311,Z 155,A 21.7149,B 23.7866,C -1.3328,E1 23.9666,E2 785.1165} C_DIS
LIN {X 120.4669,Y 58.9869,Z 155,A 23.1394,B 23.7862,C -1.3406,E1 23.9649,E2 783.6808} C_DIS
LIN {X 118.8953,Y 62.0933,Z 155,A 24.5936,B 23.7861,C -1.3431,E1 23.963,E2 782.2287} C_DIS
LIN {X 116.9317,Y 65.7198,Z 155,A 26.4513,B 23.7856,C -1.3531,E1 23.9605,E2 780.3567} C_DIS
LIN {X 114.6462,Y 69.6306,Z 155,A 28.3762,B 23.7853,C -1.3578,E1 23.9577,E2 778.4306} C_DIS
LIN {X 112.2898,Y 73.3707,Z 155,A 30.2552,B 23.7851,C -1.3623,E1 23.9549,E2 776.5505} C_DIS
LIN {X 109.828,Y 77.0068,Z 155,A 32.1496,B 23.7847,C -1.3681,E1 23.9519,E2 774.6515} C_DIS
LIN {X 107.2008,Y 80.6235,Z 155,A 34.022,B 23.7846,C -1.371,E1 23.9488,E2 772.7816} C_DIS
LIN {X 104.5135,Y 84.0777,Z 155,A 35.8673,B 23.7844,C -1.3743,E1 23.9456,E2 770.9372} C_DIS
LIN {X 101.724,Y 87.432,Z 155,A 37.7344,B 23.7842,C -1.3789,E1 23.9422,E2 769.0678} C_DIS
LIN {X 98.7308,Y 90.7983,Z 155,A 39.6102,B 23.7841,C -1.3807,E1 23.9387,E2 767.1962} C_DIS
LIN {X 95.9152,Y 93.7679,Z 155,A 41.4036,B 23.7837,C -1.387,E1 23.9352,E2 765.3955} C_DIS
LIN {X 92.6239,Y 97.0202,Z 155,A 43.3492,B 23.7836,C -1.3896,E1 23.9313,E2 763.452} C_DIS
LIN {X 89.2902,Y 100.0972,Z 155,A 45.2869,B 23.7834,C -1.3936,E1 23.9273,E2 761.5127} C_DIS
LIN {X 85.883,Y 103.0359,Z 155,A 47.231,B 23.7831,C -1.3985,E1 23.9232,E2 759.5643} C_DIS
LIN {X 82.4837,Y 105.7767,Z 155,A 49.0914,B 23.7829,C -1.4018,E1 23.9191,E2 757.7033} C_DIS
LIN {X 78.8984,Y 108.4767,Z 155,A 50.9641,B 23.7829,C -1.4029,E1 23.9149,E2 755.8348} C_DIS
LIN {X 75.4388,Y 110.9107,Z 155,A 52.7979,B 23.7826,C -1.4074,E1 23.9107,E2 753.9966} C_DIS
LIN {X 71.5267,Y 113.4727,Z 155,A 54.6007,B 23.783,C -1.4005,E1 23.9065,E2 752.217} C_DIS
LIN {X 68.3229,Y 115.4308,Z 155,A 56.3929,B 23.7823,C -1.4127,E1 23.9022,E2 750.4006} C_DIS
LIN {X 64.4369,Y 117.6438,Z 155,A 58.2687,B 23.7823,C -1.4136,E1 23.8976,E2 748.5282} C_DIS
LIN {X 61.0929,Y 119.4124,Z 155,A 59.7999,B 23.7823,C -1.4115,E1 23.8938,E2 747.0068} C_DIS
LIN {X 58.2437,Y 120.8283,Z 155,A 61.2017,B 23.7821,C -1.4154,E1 23.8903,E2 745.5993} C_DIS
LIN {X 54.8801,Y 122.3919,Z 155,A 62.7048,B 23.7823,C -1.4131,E1 23.8865,E2 744.1058} C_DIS
LIN {X 51.8324,Y 123.7135,Z 155,A 64.0722,B 23.7823,C -1.412,E1 23.883,E2 742.7445} C_DIS
LIN {X 48.7609,Y 124.956,Z 155,A 65.505,B 23.7822,C -1.4144,E1 23.8793,E2 741.3092} C_DIS
LIN {X 45.7203,Y 126.1004,Z 155,A 66.909,B 23.7821,C -1.4166,E1 23.8756,E2 739.9031} C_DIS
LIN {X 40.4434,Y 127.891,Z 155,A 69.2306,B 23.7821,C -1.4156,E1 23.8695,E2 737.5886} C_DIS
LIN {X 36.7276,Y 129.0082,Z 155,A 71.0413,B 23.7816,C -1.4246,E1 23.8646,E2 735.759} C_DIS
LIN {X 33.0637,Y 129.994,Z 155,A 72.5388,B 23.7819,C -1.4194,E1 23.8605,E2 734.2767} C_DIS
LIN {X 29.8539,Y 130.7685,Z 155,A 74.0364,B 23.7816,C -1.4246,E1 23.8564,E2 732.7684} C_DIS
LIN {X 25.5401,Y 131.6795,Z 155,A 75.9083,B 23.7816,C -1.4249,E1 23.8513,E2 730.8982} C_DIS
LIN {X 22.0208,Y 132.3131,Z 155,A 77.4048,B 23.7816,C -1.4239,E1 23.8472,E2 729.4058} C_DIS
LIN {X 17.8952,Y 132.9348,Z 155,A 79.2294,B 23.7816,C -1.4265,E1 23.8422,E2 727.5765} C_DIS
LIN {X 14.1829,Y 133.3813,Z 155,A 80.8001,B 23.7816,C -1.4255,E1 23.8378,E2 726.0095} C_DIS
LIN {X 9.9236,Y 133.7657,Z 155,A 82.6156,B 23.7816,C -1.4251,E1 23.8328,E2 724.1961} C_DIS
LIN {X 5.9853,Y 134.0017,Z 155,A 84.3775,B 23.7814,C -1.4289,E1 23.8278,E2 722.4254} C_DIS
LIN {X 2.1015,Y 134.1169,Z 155,A 85.9741,B 23.7816,C -1.4256,E1 23.8234,E2 720.8373} C_DIS
LIN {X -2.1209,Y 134.1166,Z 155,A 87.7564,B 23.7816,C -1.4241,E1 23.8184,E2 719.0586} C_DIS
LIN {X -6.0734,Y 133.9973,Z 155,A 89.5289,B 23.7814,C -1.4277,E1 23.8135,E2 717.2768} C_DIS
LIN {X -9.5824,Y 133.7906,Z 155,A 90.9583,B 23.7817,C -1.4236,E1 23.8095,E2 715.8572} C_DIS
LIN {X -13.5707,Y 133.447,Z 155,A 92.7788,B 23.7814,C -1.4282,E1 23.8044,E2 714.0242} C_DIS
LIN {X -17.3578,Y 133.0053,Z 155,A 94.2829,B 23.7818,C -1.4211,E1 23.8003,E2 712.5366} C_DIS
LIN {X -20.8886,Y 132.4971,Z 155,A 95.8793,B 23.7817,C -1.4236,E1 23.7959,E2 710.9325} C_DIS
LIN {X -25.0043,Y 131.782,Z 155,A 97.5969,B 23.7819,C -1.419,E1 23.7912,E2 709.2245} C_DIS
LIN {X -28.2512,Y 131.1241,Z 155,A 99.0225,B 23.7819,C -1.4183,E1 23.7873,E2 707.7988} C_DIS
LIN {X -31.6581,Y 130.3437,Z 155,A 100.5435,B 23.7819,C -1.4183,E1 23.7831,E2 706.2757} C_DIS
LIN {X -35.8672,Y 129.2488,Z 155,A 102.3646,B 23.7822,C -1.4146,E1 23.7782,E2 704.4608} C_DIS
LIN {X -38.9464,Y 128.3546,Z 155,A 103.7704,B 23.7822,C -1.4148,E1 23.7745,E2 703.052} C_DIS
LIN {X -42.3411,Y 127.2747,Z 155,A 105.2796,B 23.7823,C -1.4124,E1 23.7705,E2 701.5458} C_DIS
LIN {X -45.4925,Y 126.1826,Z 155,A 106.6734,B 23.7825,C -1.4091,E1 23.7668,E2 700.1573} C_DIS
LIN {X -48.8872,Y 124.9069,Z 155,A 108.3097,B 23.7824,C -1.4113,E1 23.7625,E2 698.5121} C_DIS
LIN {X -52.8821,Y 123.2689,Z 155,A 110.1345,B 23.7826,C -1.4077,E1 23.7578,E2 696.6917} C_DIS
LIN {X -56.2281,Y 121.7784,Z 155,A 111.6454,B 23.7828,C -1.4027,E1 23.754,E2 695.1893} C_DIS
LIN {X -59.29,Y 120.3174,Z 155,A 113.0709,B 23.783,C -1.3993,E1 23.7504,E2 693.7684} C_DIS
LIN {X -62.2265,Y 118.8253,Z 155,A 114.4877,B 23.7831,C -1.3974,E1 23.7469,E2 692.3522} C_DIS
LIN {X -65.7817,Y 116.8969,Z 155,A 116.3574,B 23.7829,C -1.4012,E1 23.7423,E2 690.4675} C_DIS
LIN {X -68.9474,Y 115.0586,Z 155,A 117.9537,B 23.783,C -1.3999,E1 23.7385,E2 688.8693} C_DIS
LIN {X -72.7378,Y 112.7007,Z 155,A 119.8882,B 23.7831,C -1.3976,E1 23.7339,E2 686.9341} C_DIS
LIN {X -76.5201,Y 110.1671,Z 155,A 121.7974,B 23.7834,C -1.392,E1 23.7295,E2 685.0319} C_DIS
LIN {X -81.7632,Y 106.3344,Z 155,A 125.0064,B 23.7826,C -1.407,E1 23.7223,E2 681.7736} C_DIS
LIN {X -85.1938,Y 103.6064,Z 155,A 126.5047,B 23.7838,C -1.385,E1 23.7191,E2 680.3241} C_DIS
LIN {X -91.2856,Y 98.2805,Z 155,A 130.7732,B 23.7821,C -1.4157,E1 23.7101,E2 675.9609} C_DIS
LIN {X -95.9618,Y 93.7204,Z 155,A 133.346,B 23.7831,C -1.3984,E1 23.7051,E2 673.4196} C_DIS
LIN {X -99.5939,Y 89.8513,Z 155,A 134.9289,B 23.7852,C -1.3602,E1 23.7023,E2 671.9245} C_DIS
LIN {X -102.0944,Y 86.9992,Z 155,A 136.6455,B 23.7852,C -1.3605,E1 23.6991,E2 670.1988} C_DIS
LIN {X -104.8268,Y 83.6868,Z 155,A 138.6988,B 23.7849,C -1.366,E1 23.6955,E2 668.1219} C_DIS
LIN {X -106.8198,Y 81.1283,Z 155,A 139.9358,B 23.7854,C -1.3552,E1 23.6934,E2 666.9054} C_DIS
LIN {X -109.4466,Y 77.5477,Z 155,A 141.8319,B 23.7857,C -1.35,E1 23.6904,E2 665.0127} C_DIS
LIN {X -112.0186,Y 73.7831,Z 155,A 143.77,B 23.786,C -1.344,E1 23.6874,E2 663.0792} C_DIS
LIN {X -114.4959,Y 69.8778,Z 155,A 145.7797,B 23.7863,C -1.34,E1 23.6844,E2 661.0687} C_DIS
LIN {X -116.6705,Y 66.1831,Z 155,A 147.4008,B 23.7871,C -1.3248,E1 23.6822,E2 659.4766} C_DIS
LIN {X -118.0441,Y 63.7005,Z 155,A 148.8276,B 23.7867,C -1.3312,E1 23.6802,E2 658.0258} C_DIS
LIN {X -119.9124,Y 60.1107,Z 155,A 150.8036,B 23.7864,C -1.3376,E1 23.6777,E2 656.0225} C_DIS
LIN {X -121.4181,Y 57.0075,Z 155,A 152.0687,B 23.7871,C -1.3234,E1 23.6762,E2 654.7857} C_DIS
LIN {X -122.8194,Y 53.9218,Z 155,A 153.4509,B 23.7875,C -1.3159,E1 23.6747,E2 653.4142} C_DIS
LIN {X -124.2243,Y 50.5981,Z 155,A 155.0149,B 23.7877,C -1.3122,E1 23.673,E2 651.8502} C_DIS
LIN {X -125.5279,Y 47.2696,Z 155,A 156.5106,B 23.788,C -1.306,E1 23.6715,E2 650.361} C_DIS
LIN {X -126.7992,Y 43.7448,Z 155,A 158.5816,B 23.7872,C -1.323,E1 23.6696,E2 648.2352} C_DIS
LIN {X -128.1164,Y 39.7248,Z 155,A 159.9022,B 23.7886,C -1.2945,E1 23.6685,E2 646.9777} C_DIS
LIN {X -129.2734,Y 35.7793,Z 155,A 161.7902,B 23.7886,C -1.295,E1 23.667,E2 645.0769} C_DIS
LIN {X -130.1822,Y 32.3222,Z 155,A 163.5185,B 23.7884,C -1.2995,E1 23.6659,E2 643.3267} C_DIS
LIN {X -131.4626,Y 26.6319,Z 155,A 165.7769,B 23.7893,C -1.2806,E1 23.6645,E2 641.1015} C_DIS
LIN {X -132.2463,Y 22.4212,Z 155,A 167.5917,B 23.7897,C -1.2739,E1 23.6637,E2 639.2919} C_DIS
LIN {X -132.7758,Y 19.0334,Z 155,A 169.0686,B 23.7899,C -1.2697,E1 23.663,E2 637.8162} C_DIS
LIN {X -133.2231,Y 15.6007,Z 155,A 170.5606,B 23.7901,C -1.2655,E1 23.6625,E2 636.3253} C_DIS
LIN {X -133.6332,Y 11.5746,Z 155,A 172.3137,B 23.7903,C -1.261,E1 23.6621,E2 634.5723} C_DIS
LIN {X -133.887,Y 8.1245,Z 155,A 173.8144,B 23.7905,C -1.2572,E1 23.6618,E2 633.0715} C_DIS
LIN {X -134.0775,Y 3.869,Z 155,A 175.5409,B 23.791,C -1.2469,E1 23.6616,E2 631.3596} C_DIS
LIN {X -134.133,Y 0.5663,Z 155,A 177.1085,B 23.7909,C -1.2496,E1 23.6616,E2 629.7754} C_DIS
LIN {X -134.0907,Y -3.3937,Z 155,A 178.7641,B 23.7912,C -1.2424,E1 23.6616,E2 628.1272} C_DIS
LIN {X -133.9524,Y -6.9663,Z 155,A -179.6277,B 23.7913,C -1.2412,E1 23.6619,E2 626.5117} C_DIS
LIN {X -133.6605,Y -11.2512,Z 155,A -177.8599,B 23.7917,C -1.2322,E1 23.6622,E2 624.7553} C_DIS
LIN {X -133.2774,Y -15.1449,Z 155,A -176.0708,B 23.7917,C -1.2322,E1 23.6628,E2 622.9546} C_DIS
LIN {X -132.7919,Y -18.9208,Z 155,A -174.5191,B 23.7922,C -1.2236,E1 23.6634,E2 621.4147} C_DIS
LIN {X -132.1645,Y -22.9077,Z 155,A -172.4414,B 23.7916,C -1.2347,E1 23.6643,E2 619.2964} C_DIS
LIN {X -131.5104,Y -26.3971,Z 155,A -171.1212,B 23.7923,C -1.2207,E1 23.665,E2 618.0029} C_DIS
LIN {X -130.5533,Y -30.7884,Z 155,A -169.2727,B 23.7928,C -1.2113,E1 23.6662,E2 616.1664} C_DIS
LIN {X -129.6482,Y -34.395,Z 155,A -167.6987,B 23.793,C -1.2057,E1 23.6673,E2 614.5966} C_DIS
LIN {X -128.5085,Y -38.4423,Z 155,A -165.8037,B 23.793,C -1.2048,E1 23.6688,E2 612.6923} C_DIS
LIN {X -127.3543,Y -42.102,Z 155,A -164.2887,B 23.7936,C -1.194,E1 23.6701,E2 611.1951} C_DIS
LIN {X -126.2578,Y -45.2839,Z 155,A -162.8286,B 23.7937,C -1.1907,E1 23.6714,E2 609.7344} C_DIS
LIN {X -125.0301,Y -48.5703,Z 155,A -161.3553,B 23.794,C -1.1851,E1 23.6729,E2 608.2664} C_DIS
LIN {X -123.8406,Y -51.5279,Z 155,A -159.9985,B 23.7942,C -1.1808,E1 23.6743,E2 606.9121} C_DIS
LIN {X -121.9433,Y -55.8716,Z 155,A -157.9076,B 23.7943,C -1.178,E1 23.6767,E2 604.816} C_DIS
LIN {X -120.1498,Y -59.6298,Z 155,A -156.1061,B 23.7945,C -1.1741,E1 23.6789,E2 603.0142} C_DIS
LIN {X -118.1129,Y -63.5725,Z 155,A -154.1369,B 23.7946,C -1.1722,E1 23.6815,E2 601.0385} C_DIS
LIN {X -115.9788,Y -67.3874,Z 155,A -152.2589,B 23.7948,C -1.1676,E1 23.6841,E2 599.1616} C_DIS
LIN {X -113.7195,Y -71.1343,Z 155,A -150.4049,B 23.7951,C -1.1619,E1 23.6868,E2 597.3118} C_DIS
LIN {X -111.4053,Y -74.7063,Z 155,A -148.5571,B 23.7952,C -1.1586,E1 23.6896,E2 595.4625} C_DIS
LIN {X -108.8784,Y -78.3438,Z 155,A -146.6202,B 23.7954,C -1.1559,E1 23.6927,E2 593.5222} C_DIS
LIN {X -107.1371,Y -80.7079,Z 155,A -144.8974,B 23.7945,C -1.1753,E1 23.6958,E2 591.7424} C_DIS
LIN {X -104.1768,Y -84.4951,Z 155,A -143.3066,B 23.7957,C -1.1481,E1 23.6984,E2 590.2116} C_DIS
LIN {X -101.1761,Y -88.0655,Z 155,A -141.3098,B 23.7959,C -1.1436,E1 23.702,E2 588.2162} C_DIS
LIN {X -98.0483,Y -91.5351,Z 155,A -139.3249,B 23.7961,C -1.1386,E1 23.7058,E2 586.2346} C_DIS
LIN {X -94.1294,Y -95.5602,Z 155,A -136.5933,B 23.7956,C -1.1495,E1 23.7112,E2 583.4638} C_DIS
LIN {X -91.3492,Y -98.2214,Z 155,A -135.2827,B 23.7965,C -1.1299,E1 23.7138,E2 582.1961} C_DIS
LIN {X -88.3294,Y -100.9458,Z 155,A -133.4986,B 23.7965,C -1.1287,E1 23.7176,E2 580.4077} C_DIS
LIN {X -84.882,Y -103.8612,Z 155,A -131.5755,B 23.7968,C -1.1247,E1 23.7217,E2 578.4866} C_DIS
LIN {X -81.2526,Y -106.7249,Z 155,A -129.6143,B 23.797,C -1.1204,E1 23.726,E2 576.5286} C_DIS
LIN {X -77.7029,Y -109.3367,Z 155,A -127.6859,B 23.797,C -1.1194,E1 23.7304,E2 574.5956} C_DIS
LIN {X -74.0147,Y -111.8661,Z 155,A -125.7571,B 23.797,C -1.1171,E1 23.7349,E2 572.6655} C_DIS
LIN {X -70.1761,Y -114.3128,Z 155,A -123.853,B 23.7973,C -1.1122,E1 23.7393,E2 570.7675} C_DIS
LIN {X -66.2784,Y -116.6161,Z 155,A -121.903,B 23.7974,C -1.1101,E1 23.7441,E2 568.8165} C_DIS
LIN {X -62.5976,Y -118.6305,Z 155,A -120.2095,B 23.7977,C -1.1029,E1 23.7482,E2 567.1359} C_DIS
LIN {X -59.4957,Y -120.216,Z 155,A -118.7187,B 23.7977,C -1.1011,E1 23.7519,E2 565.6452} C_DIS
LIN {X -56.4946,Y -121.6552,Z 155,A -117.2746,B 23.7978,C -1.1005,E1 23.7556,E2 564.1988} C_DIS
LIN {X -53.4018,Y -123.0442,Z 155,A -115.8236,B 23.7978,C -1.099,E1 23.7593,E2 562.7478} C_DIS
LIN {X -50.2655,Y -124.3583,Z 155,A -114.3987,B 23.798,C -1.0962,E1 23.7629,E2 561.3267} C_DIS
LIN {X -47.227,Y -125.5439,Z 155,A -112.5392,B 23.7971,C -1.118,E1 23.768,E2 559.4088} C_DIS
LIN {X -43.4474,Y -126.9024,Z 155,A -111.0766,B 23.7977,C -1.1039,E1 23.7717,E2 557.9783} C_DIS
LIN {X -39.5513,Y -128.1695,Z 155,A -109.4674,B 23.798,C -1.0955,E1 23.776,E2 556.3869} C_DIS
LIN {X -36.2682,Y -129.1366,Z 155,A -108.056,B 23.7982,C -1.092,E1 23.7797,E2 554.9818} C_DIS
LIN {X -33.4203,Y -129.9035,Z 155,A -106.729,B 23.7981,C -1.0946,E1 23.7833,E2 553.6464} C_DIS
LIN {X -29.8932,Y -130.7595,Z 155,A -105.1829,B 23.7981,C -1.0935,E1 23.7875,E2 552.1006} C_DIS
LIN {X -25.7836,Y -131.633,Z 155,A -103.3343,B 23.7981,C -1.0954,E1 23.7926,E2 550.2451} C_DIS
LIN {X -22.1151,Y -132.2974,Z 155,A -101.8504,B 23.7983,C -1.0895,E1 23.7967,E2 548.7745} C_DIS
LIN {X -18.7286,Y -132.8194,Z 155,A -100.3147,B 23.7982,C -1.0927,E1 23.8009,E2 547.2293} C_DIS
LIN {X -14.4461,Y -133.353,Z 155,A -98.5164,B 23.7982,C -1.0901,E1 23.8059,E2 545.4362} C_DIS
LIN {X -10.7329,Y -133.7043,Z 155,A -96.8029,B 23.798,C -1.0961,E1 23.8107,E2 543.707} C_DIS
LIN {X -6.6731,Y -133.9671,Z 155,A -95.1646,B 23.7982,C -1.0912,E1 23.8153,E2 542.0805} C_DIS
LIN {X -2.6233,Y -134.1082,Z 155,A -93.4004,B 23.7982,C -1.0931,E1 23.8202,E2 540.3113} C_DIS
LIN {X 0.9544,Y -134.1287,Z 155,A -92.5284,B 23.7996,C -1.0602,E1 23.8224,E2 539.5208} C_DIS
Enddeposition()
LIN {X 0.9544,Y -134.1287,Z 155,A -92.5284,B 23.7996,C -1.0602,E1 23.8224,E2 539.5208} C_DIS
Startdeposition()
$VEL.CP = VEL_PRINT
LIN {X 0.3687,Y -133.198,Z 155,A -92.5187,B 22.4298,C -0.8314,E1 22.4438,E2 539.9337} C_DIS
LIN {X -3.6264,Y -133.1486,Z 155,A -94.1297,B 22.4296,C -0.8362,E1 22.4394,E2 541.5323} C_DIS
LIN {X -7.0937,Y -133.0095,Z 155,A -95.5975,B 22.4296,C -0.8373,E1 22.4353,E2 542.9977} C_DIS
LIN {X -11.0568,Y -132.7383,Z 155,A -97.3219,B 22.4296,C -0.8366,E1 22.4305,E2 544.7246} C_DIS
LIN {X -14.4516,Y -132.4117,Z 155,A -98.7814,B 22.4296,C -0.8371,E1 22.4264,E2 546.1838} C_DIS
LIN {X -17.6504,Y -132.0236,Z 155,A -100.1807,B 22.4296,C -0.8368,E1 22.4225,E2 547.585} C_DIS
LIN {X -21.9688,Y -131.3736,Z 155,A -102.0209,B 22.4295,C -0.8391,E1 22.4175,E2 549.4209} C_DIS
LIN {X -25.1377,Y -130.8043,Z 155,A -103.4483,B 22.4295,C -0.8377,E1 22.4135,E2 550.8538} C_DIS
LIN {X -28.4555,Y -130.1232,Z 155,A -104.8774,B 22.4295,C -0.8396,E1 22.4096,E2 552.2797} C_DIS
LIN {X -31.56,Y -129.4052,Z 155,A -106.2888,B 22.4295,C -0.8385,E1 22.4058,E2 553.6963} C_DIS
LIN {X -34.6673,Y -128.6076,Z 155,A -107.6143,B 22.4295,C -0.8418,E1 22.4022,E2 555.0152} C_DIS
LIN {X -37.7743,Y -127.7295,Z 155,A -109.0664,B 22.4295,C -0.8399,E1 22.3983,E2 556.475} C_DIS
LIN {X -40.8782,Y -126.7703,Z 155,A -110.4499,B 22.4295,C -0.8416,E1 22.3946,E2 557.8568} C_DIS
LIN {X -44.4043,Y -125.5807,Z 155,A -112.0365,B 22.4293,C -0.8436,E1 22.3904,E2 559.4416} C_DIS
LIN {X -47.0644,Y -124.606,Z 155,A -113.2598,B 22.4293,C -0.8445,E1 22.3872,E2 560.6653} C_DIS
LIN {X -50.5655,Y -123.229,Z 155,A -114.8831,B 22.4293,C -0.8459,E1 22.383,E2 562.289} C_DIS
LIN {X -53.174,Y -122.1238,Z 155,A -116.1108,B 22.4293,C -0.8468,E1 22.3799,E2 563.5175} C_DIS
LIN {X -56.4769,Y -120.633,Z 155,A -117.6639,B 22.4291,C -0.8489,E1 22.3759,E2 565.0695} C_DIS
LIN {X -59.6793,Y -119.0825,Z 155,A -119.2071,B 22.4291,C -0.8502,E1 22.3721,E2 566.6139} C_DIS
LIN {X -62.6701,Y -117.536,Z 155,A -120.6612,B 22.4291,C -0.8518,E1 22.3685,E2 568.0682} C_DIS
LIN {X -66.1638,Y -115.6048,Z 155,A -122.4163,B 22.4291,C -0.8525,E1 22.3642,E2 569.8272} C_DIS
LIN {X -69.8404,Y -113.4215,Z 155,A -124.3182,B 22.4291,C -0.8525,E1 22.3596,E2 571.7359} C_DIS
LIN {X -73.601,Y -111.0187,Z 155,A -126.2748,B 22.429,C -0.8538,E1 22.355,E2 573.6961} C_DIS
LIN {X -77.1045,Y -108.6146,Z 155,A -128.0591,B 22.4288,C -0.8588,E1 22.351,E2 575.4741} C_DIS
LIN {X -80.5399,Y -106.0921,Z 155,A -129.8708,B 22.4286,C -0.863,E1 22.3469,E2 577.282} C_DIS
LIN {X -83.7849,Y -103.5481,Z 155,A -131.7089,B 22.4286,C -0.8634,E1 22.3429,E2 579.1268} C_DIS
LIN {X -87.2513,Y -100.6452,Z 155,A -133.6341,B 22.4285,C -0.8681,E1 22.3388,E2 581.0482} C_DIS
LIN {X -90.2839,Y -97.9332,Z 155,A -135.333,B 22.4282,C -0.8738,E1 22.3353,E2 582.7395} C_DIS
LIN {X -92.9597,Y -95.3979,Z 155,A -136.9263,B 22.4282,C -0.8768,E1 22.3321,E2 584.3326} C_DIS
LIN {X -95.7801,Y -92.5649,Z 155,A -138.6987,B 22.4281,C -0.8782,E1 22.3286,E2 586.1098} C_DIS
LIN {X -98.5952,Y -89.5603,Z 155,A -140.5163,B 22.4281,C -0.8801,E1 22.3252,E2 587.9315} C_DIS
LIN {X -101.4075,Y -86.3633,Z 155,A -142.3677,B 22.4279,C -0.8834,E1 22.3218,E2 589.7836} C_DIS
LIN {X -104.337,Y -82.8004,Z 155,A -144.3018,B 22.4276,C -0.8903,E1 22.3184,E2 591.7097} C_DIS
LIN {X -106.6307,Y -79.8253,Z 155,A -146.0091,B 22.4276,C -0.8903,E1 22.3155,E2 593.4263} C_DIS
LIN {X -109.2343,Y -76.2232,Z 155,A -147.9223,B 22.4274,C -0.895,E1 22.3124,E2 595.3376} C_DIS
LIN {X -111.6164,Y -72.6904,Z 155,A -149.7466,B 22.4273,C -0.9001,E1 22.3096,E2 597.1588} C_DIS
LIN {X -113.8818,Y -69.0872,Z 155,A -151.6059,B 22.4271,C -0.9037,E1 22.3069,E2 599.0193} C_DIS
LIN {X -116.208,Y -65.0985,Z 155,A -153.5294,B 22.4268,C -0.9118,E1 22.3042,E2 600.9329} C_DIS
LIN {X -118.1026,Y -61.5911,Z 155,A -155.223,B 22.4266,C -0.9174,E1 22.302,E2 602.6218} C_DIS
LIN {X -119.6195,Y -58.5907,Z 155,A -156.6775,B 22.4264,C -0.9211,E1 22.3002,E2 604.0754} C_DIS
LIN {X -121.0543,Y -55.5658,Z 155,A -158.1256,B 22.4263,C -0.9248,E1 22.2985,E2 605.5226} C_DIS
LIN {X -122.4067,Y -52.5195,Z 155,A -159.5616,B 22.4261,C -0.9289,E1 22.2969,E2 606.9568} C_DIS
LIN {X -123.6765,Y -49.4552,Z 155,A -161.0408,B 22.4261,C -0.9307,E1 22.2953,E2 608.4405} C_DIS
LIN {X -125.0237,Y -45.9492,Z 155,A -162.6277,B 22.4258,C -0.9367,E1 22.2937,E2 610.0217} C_DIS
LIN {X -125.9109,Y -43.4518,Z 155,A -163.7698,B 22.4258,C -0.94,E1 22.2927,E2 611.1623} C_DIS
LIN {X -126.9562,Y -40.2963,Z 155,A -165.2266,B 22.4256,C -0.9432,E1 22.2914,E2 612.6203} C_DIS
LIN {X -128.0584,Y -36.6511,Z 155,A -166.8602,B 22.4254,C -0.9483,E1 22.2901,E2 614.251} C_DIS
LIN {X -128.8063,Y -33.9223,Z 155,A -168.0786,B 22.4252,C -0.952,E1 22.2893,E2 615.4677} C_DIS
LIN {X -129.676,Y -30.4369,Z 155,A -169.6383,B 22.4251,C -0.9561,E1 22.2882,E2 617.0269} C_DIS
LIN {X -130.3653,Y -27.334,Z 155,A -171.0134,B 22.4249,C -0.96,E1 22.2874,E2 618.4007} C_DIS
LIN {X -130.9763,Y -24.2375,Z 155,A -172.3789,B 22.4247,C -0.9639,E1 22.2867,E2 619.7651} C_DIS
LIN {X -131.4858,Y -21.2966,Z 155,A -173.6397,B 22.4245,C -0.969,E1 22.2861,E2 621.0211} C_DIS
LIN {X -131.9073,Y -18.4999,Z 155,A -174.9294,B 22.4245,C -0.9697,E1 22.2856,E2 622.3176} C_DIS
LIN {X -132.3008,Y -15.4365,Z 155,A -176.2294,B 22.4243,C -0.9751,E1 22.2852,E2 623.612} C_DIS
LIN {X -132.6209,Y -12.3894,Z 155,A -177.5548,B 22.4241,C -0.979,E1 22.2848,E2 624.9362} C_DIS
LIN {X -132.869,Y -9.3609,Z 155,A -178.8581,B 22.4239,C -0.9833,E1 22.2845,E2 626.2369} C_DIS
LIN {X -133.0468,Y -6.3532,Z 155,A 179.7926,B 22.4239,C -0.9852,E1 22.2843,E2 627.5904} C_DIS
LIN {X -133.1558,Y -3.3683,Z 155,A 178.5139,B 22.4237,C -0.9896,E1 22.2842,E2 628.8661} C_DIS
LIN {X -133.201,Y 0,Z 155,A 177.0449,B 22.4235,C -0.9934,E1 22.2842,E2 630.3353} C_DIS
LIN {X -133.1558,Y 3.3683,Z 155,A 175.5373,B 22.4235,C -0.9956,E1 22.2842,E2 631.8473} C_DIS
LIN {X -133.026,Y 6.767,Z 155,A 174.1193,B 22.4231,C -1.0022,E1 22.2844,E2 633.2574} C_DIS
LIN {X -132.8293,Y 9.9051,Z 155,A 172.7137,B 22.4231,C -1.0043,E1 22.2847,E2 634.667} C_DIS
LIN {X -132.5153,Y 13.4887,Z 155,A 171.2089,B 22.4228,C -1.0111,E1 22.2851,E2 636.1642} C_DIS
LIN {X -132.1689,Y 16.542,Z 155,A 169.8749,B 22.4226,C -1.0148,E1 22.2855,E2 637.4974} C_DIS
LIN {X -131.5762,Y 20.7241,Z 155,A 168.0403,B 22.4224,C -1.0199,E1 22.2863,E2 639.3308} C_DIS
LIN {X -131.0529,Y 23.8098,Z 155,A 166.6819,B 22.4222,C -1.0237,E1 22.2869,E2 640.6883} C_DIS
LIN {X -130.4526,Y 26.9051,Z 155,A 165.3129,B 22.4221,C -1.0275,E1 22.2877,E2 642.0565} C_DIS
LIN {X -129.7741,Y 30.0072,Z 155,A 163.9345,B 22.4219,C -1.0313,E1 22.2885,E2 643.434} C_DIS
LIN {X -128.9935,Y 33.2039,Z 155,A 162.5187,B 22.4217,C -1.0358,E1 22.2895,E2 644.8474} C_DIS
LIN {X -128.0584,Y 36.6511,Z 155,A 160.9569,B 22.4215,C -1.0395,E1 22.2906,E2 646.4095} C_DIS
LIN {X -127.1286,Y 39.7566,Z 155,A 159.5503,B 22.4214,C -1.0433,E1 22.2918,E2 647.8151} C_DIS
LIN {X -126.1172,Y 42.857,Z 155,A 158.1353,B 22.4212,C -1.0472,E1 22.293,E2 649.2291} C_DIS
LIN {X -124.6374,Y 46.9805,Z 155,A 156.2232,B 22.421,C -1.0519,E1 22.2949,E2 651.1411} C_DIS
LIN {X -123.229,Y 50.5655,Z 155,A 154.5641,B 22.4208,C -1.0568,E1 22.2966,E2 652.7977} C_DIS
LIN {X -121.9293,Y 53.6238,Z 155,A 153.1228,B 22.4206,C -1.0606,E1 22.2982,E2 654.2379} C_DIS
LIN {X -120.5471,Y 56.6627,Z 155,A 151.6752,B 22.4204,C -1.0644,E1 22.2999,E2 655.6843} C_DIS
LIN {X -119.0825,Y 59.6793,Z 155,A 150.2214,B 22.4203,C -1.0682,E1 22.3017,E2 657.1371} C_DIS
LIN {X -117.536,Y 62.6701,Z 155,A 148.8543,B 22.4199,C -1.0759,E1 22.3034,E2 658.492} C_DIS
LIN {X -115.971,Y 65.5201,Z 155,A 147.2774,B 22.4201,C -1.0723,E1 22.3056,E2 660.0877} C_DIS
LIN {X -113.7601,Y 69.2885,Z 155,A 145.3277,B 22.42,C -1.0747,E1 22.3084,E2 662.0425} C_DIS
LIN {X -111.4879,Y 72.8884,Z 155,A 143.4906,B 22.4197,C -1.0796,E1 22.3112,E2 663.8773} C_DIS
LIN {X -109.0936,Y 76.4254,Z 155,A 141.6304,B 22.4196,C -1.0836,E1 22.3141,E2 665.7372} C_DIS
LIN {X -106.4369,Y 80.0831,Z 155,A 139.6985,B 22.4193,C -1.0894,E1 22.3173,E2 667.6642} C_DIS
LIN {X -103.8006,Y 83.4719,Z 155,A 137.8393,B 22.4191,C -1.0938,E1 22.3205,E2 669.5219} C_DIS
LIN {X -101.0515,Y 86.7796,Z 155,A 136.0112,B 22.4188,C -1.0995,E1 22.3238,E2 671.3445} C_DIS
LIN {X -98.5152,Y 89.6485,Z 155,A 134.4282,B 22.4185,C -1.1064,E1 22.3267,E2 672.9172} C_DIS
LIN {X -95.9643,Y 92.3747,Z 155,A 132.6923,B 22.4185,C -1.1047,E1 22.3301,E2 674.6661} C_DIS
LIN {X -92.9597,Y 95.3979,Z 155,A 130.9689,B 22.4181,C -1.1138,E1 22.3335,E2 676.3736} C_DIS
LIN {X -90.4596,Y 97.7718,Z 155,A 129.4779,B 22.4181,C -1.1169,E1 22.3365,E2 677.8633} C_DIS
LIN {X -87.9001,Y 100.0791,Z 155,A 127.9881,B 22.4179,C -1.12,E1 22.3396,E2 679.3517} C_DIS
LIN {X -84.805,Y 102.7143,Z 155,A 126.1995,B 22.4178,C -1.1221,E1 22.3435,E2 681.1426} C_DIS
LIN {X -81.7509,Y 105.1613,Z 155,A 124.4319,B 22.4178,C -1.1221,E1 22.3473,E2 682.9178} C_DIS
LIN {X -78.1812,Y 107.8415,Z 155,A 122.5433,B 22.4175,C -1.1273,E1 22.3516,E2 684.7999} C_DIS
LIN {X -74.8227,Y 110.1983,Z 155,A 120.7317,B 22.4175,C -1.1288,E1 22.3557,E2 686.6147} C_DIS
LIN {X -71.2563,Y 112.5374,Z 155,A 118.8904,B 22.4173,C -1.1319,E1 22.3601,E2 688.4544} C_DIS
LIN {X -67.3308,Y 114.929,Z 155,A 116.9224,B 22.4171,C -1.1359,E1 22.3648,E2 690.4187} C_DIS
LIN {X -63.4134,Y 117.1367,Z 155,A 114.9463,B 22.4171,C -1.1374,E1 22.3696,E2 692.3973} C_DIS
LIN {X -60.0942,Y 118.8713,Z 155,A 113.458,B 22.4166,C -1.1454,E1 22.3733,E2 693.8691} C_DIS
LIN {X -57.1586,Y 120.3102,Z 155,A 112.0453,B 22.4166,C -1.1473,E1 22.3768,E2 695.2809} C_DIS
LIN {X -54.1529,Y 121.6926,Z 155,A 110.6049,B 22.4165,C -1.1487,E1 22.3805,E2 696.7216} C_DIS
LIN {X -50.5655,Y 123.229,Z 155,A 108.9369,B 22.4163,C -1.1515,E1 22.3848,E2 698.3866} C_DIS
LIN {X -47.4913,Y 124.4461,Z 155,A 107.512,B 22.4163,C -1.1532,E1 22.3885,E2 699.8103} C_DIS
LIN {X -44.832,Y 125.4265,Z 155,A 106.2908,B 22.4162,C -1.1547,E1 22.3917,E2 701.0304} C_DIS
LIN {X -41.7365,Y 126.4903,Z 155,A 104.843,B 22.4162,C -1.1547,E1 22.3955,E2 702.4815} C_DIS
LIN {X -38.634,Y 127.4721,Z 155,A 103.4446,B 22.4162,C -1.1562,E1 22.3992,E2 703.8784} C_DIS
LIN {X -34.1858,Y 128.736,Z 155,A 101.4709,B 22.416,C -1.159,E1 22.4045,E2 705.8484} C_DIS
LIN {X -30.4369,Y 129.676,Z 155,A 99.824,B 22.4159,C -1.1612,E1 22.409,E2 707.4921} C_DIS
LIN {X -27.334,Y 130.3653,Z 155,A 98.4562,B 22.4159,C -1.1623,E1 22.4127,E2 708.8588} C_DIS
LIN {X -24.2375,Y 130.9763,Z 155,A 97.0982,B 22.4158,C -1.1633,E1 22.4165,E2 710.2158} C_DIS
LIN {X -20.3081,Y 131.6406,Z 155,A 95.3894,B 22.4157,C -1.1648,E1 22.4212,E2 711.9225} C_DIS
LIN {X -17.0541,Y 132.1018,Z 155,A 93.985,B 22.4157,C -1.1661,E1 22.425,E2 713.3248} C_DIS
LIN {X -13.9108,Y 132.4699,Z 155,A 92.6106,B 22.4157,C -1.1661,E1 22.4289,E2 714.6998} C_DIS
LIN {X -10.4532,Y 132.7893,Z 155,A 90.9511,B 22.416,C -1.1593,E1 22.4335,E2 716.3783} C_DIS
LIN {X -6.6668,Y 133.031,Z 155,A 89.4587,B 22.4156,C -1.1663,E1 22.4376,E2 717.8529} C_DIS
LIN {X -3.3683,Y 133.1558,Z 155,A 87.9314,B 22.4158,C -1.1617,E1 22.4419,E2 719.3923} C_DIS
LIN {X 0.7323,Y 133.196,Z 155,A 86.2524,B 22.4156,C -1.1659,E1 22.4466,E2 721.0603} C_DIS
LIN {X 4.4443,Y 133.1259,Z 155,A 84.6033,B 22.4157,C -1.1637,E1 22.4512,E2 722.7149} C_DIS
LIN {X 8.116,Y 132.9505,Z 155,A 83.0768,B 22.4157,C -1.1662,E1 22.4554,E2 724.2341} C_DIS
LIN {X 11.4777,Y 132.7027,Z 155,A 81.6529,B 22.4156,C -1.1673,E1 22.4594,E2 725.6544} C_DIS
LIN {X 15.0133,Y 132.3513,Z 155,A 80.1376,B 22.4156,C -1.1676,E1 22.4636,E2 727.1678} C_DIS
LIN {X 17.6504,Y 132.0236,Z 155,A 78.983,B 22.4156,C -1.1668,E1 22.4668,E2 728.3233} C_DIS
LIN {X 20.7032,Y 131.5794,Z 155,A 77.6794,B 22.4156,C -1.1675,E1 22.4704,E2 729.6239} C_DIS
LIN {X 23.5536,Y 131.0987,Z 155,A 76.407,B 22.4156,C -1.1657,E1 22.4739,E2 730.8994} C_DIS
LIN {X 26.6862,Y 130.4971,Z 155,A 75.0155,B 22.4157,C -1.1641,E1 22.4777,E2 732.293} C_DIS
LIN {X 30.0072,Y 129.7741,Z 155,A 73.5845,B 22.4157,C -1.1648,E1 22.4816,E2 733.7202} C_DIS
LIN {X 32.9485,Y 129.0583,Z 155,A 72.2712,B 22.4157,C -1.1635,E1 22.4852,E2 735.0347} C_DIS
LIN {X 36.5323,Y 128.0916,Z 155,A 70.6982,B 22.4157,C -1.1635,E1 22.4894,E2 736.6048} C_DIS
LIN {X 39.3278,Y 127.2598,Z 155,A 69.4321,B 22.4158,C -1.162,E1 22.4928,E2 737.8723} C_DIS
LIN {X 42.857,Y 126.1172,Z 155,A 67.8379,B 22.4158,C -1.1606,E1 22.497,E2 739.4665} C_DIS
LIN {X 45.9492,Y 125.0237,Z 155,A 66.4283,B 22.416,C -1.1594,E1 22.5007,E2 740.8761} C_DIS
LIN {X 48.6042,Y 124.0135,Z 155,A 65.2063,B 22.416,C -1.1582,E1 22.5039,E2 742.0982} C_DIS
LIN {X 51.6088,Y 122.7933,Z 155,A 63.7818,B 22.4162,C -1.1553,E1 22.5076,E2 743.5265} C_DIS
LIN {X 54.8725,Y 121.3708,Z 155,A 62.268,B 22.4162,C -1.1544,E1 22.5114,E2 745.0385} C_DIS
LIN {X 58.0569,Y 119.881,Z 155,A 60.7839,B 22.4162,C -1.1538,E1 22.5152,E2 746.5197} C_DIS
LIN {X 61.1781,Y 118.3195,Z 155,A 59.2782,B 22.4163,C -1.1517,E1 22.5189,E2 748.0265} C_DIS
LIN {X 63.6186,Y 117.0247,Z 155,A 57.9875,B 22.4167,C -1.1452,E1 22.5221,E2 749.3299} C_DIS
LIN {X 67.3034,Y 114.9451,Z 155,A 56.1718,B 22.4167,C -1.1427,E1 22.5265,E2 751.1458} C_DIS
LIN {X 71.1976,Y 112.5744,Z 155,A 54.2794,B 22.4167,C -1.143,E1 22.531,E2 753.0309} C_DIS
LIN {X 74.8399,Y 110.1867,Z 155,A 52.3673,B 22.417,C -1.138,E1 22.5355,E2 754.9486} C_DIS
LIN {X 78.5149,Y 107.5995,Z 155,A 50.4711,B 22.417,C -1.1365,E1 22.5398,E2 756.8414} C_DIS
LIN {X 81.9388,Y 105.0157,Z 155,A 48.6301,B 22.4172,C -1.1333,E1 22.5438,E2 758.6831} C_DIS
LIN {X 85.2054,Y 102.3827,Z 155,A 46.7994,B 22.4174,C -1.1286,E1 22.5478,E2 760.5181} C_DIS
LIN {X 88.574,Y 99.483,Z 155,A 44.8679,B 22.4177,C -1.1239,E1 22.5519,E2 762.4535} C_DIS
LIN {X 91.5436,Y 96.7568,Z 155,A 43.2362,B 22.4177,C -1.1252,E1 22.5552,E2 764.0741} C_DIS
LIN {X 94.1867,Y 94.1867,Z 155,A 41.6024,B 22.4179,C -1.1195,E1 22.5584,E2 765.7151} C_DIS
LIN {X 97.1845,Y 91.0902,Z 155,A 39.8409,B 22.4179,C -1.1199,E1 22.5618,E2 767.4669} C_DIS
LIN {X 99.5086,Y 88.5454,Z 155,A 38.2841,B 22.4182,C -1.1129,E1 22.5648,E2 769.0341} C_DIS
LIN {X 102.3175,Y 85.2841,Z 155,A 36.3949,B 22.4185,C -1.1067,E1 22.5682,E2 770.9298} C_DIS
LIN {X 105.0157,Y 81.9388,Z 155,A 34.6053,B 22.4185,C -1.1052,E1 22.5713,E2 772.714} C_DIS
LIN {X 107.5995,Y 78.5149,Z 155,A 32.7239,B 22.4189,C -1.0988,E1 22.5744,E2 774.6017} C_DIS
LIN {X 110.189,Y 74.8365,Z 155,A 30.8218,B 22.419,C -1.0955,E1 22.5774,E2 776.502} C_DIS
LIN {X 112.7406,Y 70.9342,Z 155,A 28.8587,B 22.4192,C -1.0923,E1 22.5804,E2 778.4622} C_DIS
LIN {X 115.064,Y 67.1009,Z 155,A 26.8956,B 22.4195,C -1.0854,E1 22.5832,E2 780.4319} C_DIS
LIN {X 117.1367,Y 63.4134,Z 155,A 25.0933,B 22.4197,C -1.0813,E1 22.5856,E2 782.2343} C_DIS
LIN {X 118.8374,Y 60.1607,Z 155,A 23.6552,B 22.4195,C -1.0839,E1 22.5874,E2 783.6571} C_DIS
LIN {X 120.3472,Y 57.0811,Z 155,A 22.186,B 22.4197,C -1.08,E1 22.5892,E2 785.1275} C_DIS
LIN {X 121.7408,Y 54.0451,Z 155,A 20.7601,B 22.4199,C -1.0764,E1 22.5909,E2 786.554} C_DIS
LIN {X 123.1059,Y 50.8602,Z 155,A 19.2922,B 22.42,C -1.0732,E1 22.5925,E2 788.0212} C_DIS
LIN {X 124.3661,Y 47.6971,Z 155,A 17.8258,B 22.4202,C -1.0688,E1 22.594,E2 789.4899} C_DIS
LIN {X 125.3904,Y 44.9321,Z 155,A 16.557,B 22.4204,C -1.0651,E1 22.5952,E2 790.7605} C_DIS
LIN {X 126.4903,Y 41.7365,Z 155,A 15.0908,B 22.4206,C -1.0601,E1 22.5965,E2 792.2302} C_DIS
LIN {X 127.4721,Y 38.634,Z 155,A 13.7029,B 22.4208,C -1.0564,E1 22.5976,E2 793.6187} C_DIS
LIN {X 128.3726,Y 35.5275,Z 155,A 12.3696,B 22.4208,C -1.0551,E1 22.5986,E2 794.9471} C_DIS
LIN {X 129.1924,Y 32.42,Z 155,A 10.9534,B 22.4211,C -1.0491,E1 22.5996,E2 796.3695} C_DIS
LIN {X 130.0305,Y 28.8848,Z 155,A 9.4405,B 22.4212,C -1.0467,E1 22.6006,E2 797.8788} C_DIS
LIN {X 130.6806,Y 25.7847,Z 155,A 8.0898,B 22.4214,C -1.0431,E1 22.6013,E2 799.2301} C_DIS
LIN {X 131.1595,Y 23.2142,Z 155,A 6.9948,B 22.4214,C -1.0411,E1 22.6019,E2 800.3231} C_DIS
LIN {X 131.6533,Y 20.2261,Z 155,A 5.6586,B 22.4217,C -1.0353,E1 22.6025,E2 801.6655} C_DIS
LIN {X 132.1689,Y 16.542,Z 155,A 4.0986,B 22.4219,C -1.0322,E1 22.603,E2 803.2232} C_DIS
LIN {X 132.4699,Y 13.9108,Z 155,A 2.9373,B 22.4221,C -1.0275,E1 22.6034,E2 804.389} C_DIS
LIN {X 132.8246,Y 9.9687,Z 155,A 1.2218,B 22.4223,C -1.0214,E1 22.6038,E2 806.1089} C_DIS
LIN {X 133.0363,Y 6.5607,Z 155,A -0.2412,B 22.4225,C -1.017,E1 22.604,E2 807.5737} C_DIS
LIN {X 133.1817,Y 2.086,Z 155,A -2.0633,B 22.4225,C -1.0159,E1 22.6042,E2 809.3862} C_DIS
LIN {X 133.195,Y -1.0147,Z 155,A -3.5797,B 22.4231,C -1.0025,E1 22.6042,E2 810.9273} C_DIS
LIN {X 133.1008,Y -5.0867,Z 155,A -5.188,B 22.4231,C -1.004,E1 22.604,E2 812.5209} C_DIS
LIN {X 132.9252,Y -8.5262,Z 155,A -6.6548,B 22.4232,C -1,E1 22.6038,E2 813.9885} C_DIS
LIN {X 132.6613,Y -11.9686,Z 155,A -8.0966,B 22.4234,C -0.9973,E1 22.6034,E2 815.4275} C_DIS
LIN {X 132.245,Y -15.9041,Z 155,A -9.8068,B 22.4236,C -0.9914,E1 22.6029,E2 817.1416} C_DIS
LIN {X 131.8335,Y -19.0165,Z 155,A -11.1223,B 22.4237,C -0.9888,E1 22.6024,E2 818.4552} C_DIS
LIN {X 131.3241,Y -22.2656,Z 155,A -12.5392,B 22.4239,C -0.9842,E1 22.6018,E2 819.8748} C_DIS
LIN {X 130.7624,Y -25.3564,Z 155,A -13.8827,B 22.4241,C -0.9802,E1 22.6011,E2 821.2197} C_DIS
LIN {X 130.1232,Y -28.4555,Z 155,A -15.2142,B 22.4241,C -0.9773,E1 22.6003,E2 822.5499} C_DIS
LIN {X 129.4143,Y -31.5223,Z 155,A -16.5794,B 22.4244,C -0.9725,E1 22.5994,E2 823.919} C_DIS
LIN {X 128.6557,Y -34.487,Z 155,A -17.8929,B 22.4246,C -0.9684,E1 22.5985,E2 825.2344} C_DIS
LIN {X 127.7295,Y -37.7743,Z 155,A -19.3878,B 22.4248,C -0.9625,E1 22.5973,E2 826.735} C_DIS
LIN {X 126.7703,Y -40.8782,Z 155,A -20.7454,B 22.4248,C -0.9601,E1 22.5962,E2 828.0903} C_DIS
LIN {X 125.6935,Y -44.0789,Z 155,A -22.2066,B 22.4251,C -0.9552,E1 22.5949,E2 829.555} C_DIS
LIN {X 124.606,Y -47.0644,Z 155,A -23.5427,B 22.4252,C -0.9525,E1 22.5936,E2 830.8897} C_DIS
LIN {X 123.229,Y -50.5655,Z 155,A -25.1507,B 22.4254,C -0.948,E1 22.5919,E2 832.4994} C_DIS
LIN {X 121.9293,Y -53.6238,Z 155,A -26.5716,B 22.4255,C -0.9441,E1 22.5903,E2 833.9218} C_DIS
LIN {X 120.7503,Y -56.2231,Z 155,A -27.8067,B 22.4257,C -0.94,E1 22.5889,E2 835.1599} C_DIS
LIN {X 119.2998,Y -59.2387,Z 155,A -29.2655,B 22.4259,C -0.9348,E1 22.5871,E2 836.6235} C_DIS
LIN {X 117.2472,Y -63.2076,Z 155,A -31.2226,B 22.4262,C -0.9273,E1 22.5845,E2 838.5884} C_DIS
LIN {X 115.064,Y -67.1009,Z 155,A -33.1709,B 22.4265,C -0.9203,E1 22.5818,E2 840.5435} C_DIS
LIN {X 112.866,Y -70.7356,Z 155,A -34.9876,B 22.4267,C -0.9156,E1 22.5792,E2 842.362} C_DIS
LIN {X 110.4226,Y -74.4914,Z 155,A -36.8844,B 22.4268,C -0.9118,E1 22.5762,E2 844.2583} C_DIS
LIN {X 107.9631,Y -78.0133,Z 155,A -38.7174,B 22.427,C -0.9074,E1 22.5733,E2 846.0925} C_DIS
LIN {X 105.1613,Y -81.7509,Z 155,A -40.6839,B 22.4271,C -0.9041,E1 22.5699,E2 848.0571} C_DIS
LIN {X 102.4538,Y -85.1195,Z 155,A -42.5442,B 22.4273,C -0.8992,E1 22.5667,E2 849.9206} C_DIS
LIN {X 99.6665,Y -88.3668,Z 155,A -44.2875,B 22.4273,C -0.8992,E1 22.5635,E2 851.6548} C_DIS
LIN {X 97.1845,Y -91.0902,Z 155,A -45.9383,B 22.4276,C -0.892,E1 22.5603,E2 853.3162} C_DIS
LIN {X 94.1867,Y -94.1867,Z 155,A -47.8138,B 22.4278,C -0.8864,E1 22.5566,E2 855.1973} C_DIS
LIN {X 91.0902,Y -97.1845,Z 155,A -49.5505,B 22.4278,C -0.8878,E1 22.5532,E2 856.9224} C_DIS
LIN {X 88.5454,Y -99.5086,Z 155,A -51.1556,B 22.4281,C -0.8783,E1 22.5498,E2 858.5448} C_DIS
LIN {X 85.202,Y -102.3855,Z 155,A -53.0345,B 22.4281,C -0.875,E1 22.5458,E2 860.4243} C_DIS
LIN {X 81.7509,Y -105.1613,Z 155,A -54.9131,B 22.4283,C -0.8722,E1 22.5417,E2 862.3023} C_DIS
LIN {X 78.0133,Y -107.9631,Z 155,A -56.8364,B 22.4283,C -0.8722,E1 22.5374,E2 864.2178} C_DIS
LIN {X 74.5032,Y -110.4146,Z 155,A -58.7271,B 22.4285,C -0.8661,E1 22.533,E2 866.1172} C_DIS
LIN {X 70.7356,Y -112.866,Z 155,A -60.6205,B 22.4285,C -0.8643,E1 22.5285,E2 868.0082} C_DIS
LIN {X 67.1213,Y -115.052,Z 155,A -62.4795,B 22.4288,C -0.859,E1 22.5241,E2 869.8747} C_DIS
LIN {X 63.4134,Y -117.1367,Z 155,A -64.3148,B 22.4289,C -0.8555,E1 22.5196,E2 871.713} C_DIS
LIN {X 60.0942,Y -118.8713,Z 155,A -65.7936,B 22.4288,C -0.8593,E1 22.5159,E2 873.1774} C_DIS
LIN {X 57.1872,Y -120.2965,Z 155,A -67.1943,B 22.4288,C -0.8567,E1 22.5124,E2 874.5808} C_DIS
LIN {X 54.0721,Y -121.7288,Z 155,A -68.6421,B 22.4289,C -0.8557,E1 22.5087,E2 876.027} C_DIS
LIN {X 50.8714,Y -123.1013,Z 155,A -70.1289,B 22.4289,C -0.8541,E1 22.5049,E2 877.514} C_DIS
LIN {X 47.4913,Y -124.4461,Z 155,A -71.6976,B 22.429,C -0.8517,E1 22.5008,E2 879.085} C_DIS
LIN {X 44.832,Y -125.4265,Z 155,A -72.9115,B 22.429,C -0.8504,E1 22.4976,E2 880.2994} C_DIS
LIN {X 41.7365,Y -126.4903,Z 155,A -74.351,B 22.4292,C -0.8472,E1 22.4938,E2 881.7443} C_DIS
LIN {X 38.634,Y -127.4721,Z 155,A -75.745,B 22.4292,C -0.8458,E1 22.4901,E2 883.1389} C_DIS
LIN {X 35.5275,Y -128.3726,Z 155,A -77.1305,B 22.4293,C -0.8446,E1 22.4864,E2 884.525} C_DIS
LIN {X 32.42,Y -129.1924,Z 155,A -78.4566,B 22.4293,C -0.8459,E1 22.4828,E2 885.8455} C_DIS
LIN {X 29.3032,Y -129.9349,Z 155,A -79.8499,B 22.4293,C -0.8439,E1 22.479,E2 887.2419} C_DIS
LIN {X 25.7847,Y -130.6806,Z 155,A -81.3859,B 22.4293,C -0.8431,E1 22.4748,E2 888.7779} C_DIS
LIN {X 23.1105,Y -131.178,Z 155,A -82.5859,B 22.4294,C -0.8408,E1 22.4715,E2 889.9824} C_DIS
LIN {X 19.6108,Y -131.7485,Z 155,A -84.2002,B 22.4296,C -0.8354,E1 22.467,E2 891.6089} C_DIS
LIN {X 15.8682,Y -132.2493,Z 155,A -85.7134,B 22.4295,C -0.8397,E1 22.4628,E2 893.1095} C_DIS
LIN {X 12.5807,Y -132.6025,Z 155,A -87.132,B 22.4295,C -0.8391,E1 22.4589,E2 894.5286} C_DIS
LIN {X 9.3609,Y -132.869,Z 155,A -88.5165,B 22.4295,C -0.8387,E1 22.455,E2 895.9134} C_DIS
LIN {X 6.2385,Y -133.0525,Z 155,A -89.9961,B 22.4298,C -0.8319,E1 22.4509,E2 897.4103} C_DIS
LIN {X 2.1674,Y -133.1804,Z 155,A -91.6307,B 22.4296,C -0.8369,E1 22.4463,E2 899.0314} C_DIS
LIN {X 2.1674,Y -133.1804,Z 155,A -91.6307,B 22.4296,C -0.8369,E1 22.4463,E2 899.0314} C_DIS
Enddeposition()
LIN {X 0.935,Y -132.2575,Z 155,A -91.3207,B 21.3951,C -0.7116,E1 21.4086,E2 898.9431} C_DIS
Startdeposition()
$VEL.CP = VEL_PRINT
LIN {X 4.2536,Y -132.1956,Z 155,A -89.6439,B 21.3948,C -0.7227,E1 21.4134,E2 897.2362} C_DIS
LIN {X 8.4018,Y -131.9958,Z 155,A -87.8789,B 21.3948,C -0.7219,E1 21.4183,E2 895.4744} C_DIS
LIN {X 12.528,Y -131.668,Z 155,A -86.1611,B 21.3948,C -0.7194,E1 21.423,E2 893.7647} C_DIS
LIN {X 16.106,Y -131.279,Z 155,A -84.5082,B 21.3948,C -0.7245,E1 21.4276,E2 892.0992} C_DIS
LIN {X 20.7745,Y -130.6219,Z 155,A -82.6281,B 21.3949,C -0.7185,E1 21.4328,E2 890.2376} C_DIS
LIN {X 23.58,Y -130.1439,Z 155,A -81.0882,B 21.3944,C -0.7334,E1 21.4371,E2 888.6587} C_DIS
LIN {X 27.8324,Y -129.3009,Z 155,A -79.4574,B 21.3948,C -0.7237,E1 21.4415,E2 887.057} C_DIS
LIN {X 31.2936,Y -128.5074,Z 155,A -77.8835,B 21.3947,C -0.7268,E1 21.4458,E2 885.4773} C_DIS
LIN {X 34.6293,Y -127.6498,Z 155,A -76.4575,B 21.3947,C -0.7253,E1 21.4496,E2 884.0582} C_DIS
LIN {X 38.3654,Y -126.5762,Z 155,A -74.7156,B 21.3946,C -0.7298,E1 21.4543,E2 882.3075} C_DIS
LIN {X 41.3217,Y -125.6426,Z 155,A -73.351,B 21.3945,C -0.7323,E1 21.458,E2 880.939} C_DIS
LIN {X 44.771,Y -124.4543,Z 155,A -71.8728,B 21.3945,C -0.7296,E1 21.4618,E2 879.4717} C_DIS
LIN {X 48.7889,Y -122.9368,Z 155,A -70.0476,B 21.3945,C -0.7305,E1 21.4666,E2 877.649} C_DIS
LIN {X 50.9664,Y -122.048,Z 155,A -68.9642,B 21.3944,C -0.7349,E1 21.4694,E2 876.5565} C_DIS
LIN {X 54.1657,Y -120.6623,Z 155,A -67.4649,B 21.3944,C -0.7366,E1 21.4732,E2 875.0568} C_DIS
LIN {X 57.3859,Y -119.1651,Z 155,A -65.9268,B 21.3943,C -0.739,E1 21.4771,E2 873.5171} C_DIS
LIN {X 61.6051,Y -117.0389,Z 155,A -64.0484,B 21.3944,C -0.7345,E1 21.4817,E2 871.657} C_DIS
LIN {X 64.6451,Y -115.39,Z 155,A -62.2988,B 21.3939,C -0.7487,E1 21.4861,E2 869.8746} C_DIS
LIN {X 68.6241,Y -113.0689,Z 155,A -60.3076,B 21.3939,C -0.7522,E1 21.4909,E2 867.8814} C_DIS
LIN {X 72.4672,Y -110.6454,Z 155,A -58.4074,B 21.3939,C -0.7527,E1 21.4953,E2 865.9871} C_DIS
LIN {X 75.9492,Y -108.285,Z 155,A -56.1121,B 21.3929,C -0.7786,E1 21.5007,E2 863.6305} C_DIS
LIN {X 79.5751,Y -105.6485,Z 155,A -54.6643,B 21.3936,C -0.7593,E1 21.5038,E2 862.2415} C_DIS
LIN {X 82.857,Y -103.0949,Z 155,A -52.8247,B 21.3934,C -0.7649,E1 21.5079,E2 860.3947} C_DIS
LIN {X 87.5867,Y -99.1078,Z 155,A -50.0629,B 21.3931,C -0.7748,E1 21.5138,E2 857.6189} C_DIS
LIN {X 91.2548,Y -95.7412,Z 155,A -48.0314,B 21.3931,C -0.7739,E1 21.5179,E2 855.5997} C_DIS
LIN {X 94.3528,Y -92.6895,Z 155,A -45.8621,B 21.3925,C -0.7919,E1 21.5222,E2 853.3921} C_DIS
LIN {X 96.9027,Y -90.0205,Z 155,A -43.9497,B 21.3918,C -0.8109,E1 21.5259,E2 851.4381} C_DIS
LIN {X 100.4978,Y -85.9893,Z 155,A -42.4931,B 21.3931,C -0.7747,E1 21.5284,E2 850.0878} C_DIS
LIN {X 103.3901,Y -82.4882,Z 155,A -39.3905,B 21.3909,C -0.8341,E1 21.5341,E2 846.8405} C_DIS
LIN {X 107.5101,Y -77.0415,Z 155,A -37.5141,B 21.3925,C -0.7902,E1 21.5369,E2 845.0946} C_DIS
LIN {X 109.6083,Y -74.0259,Z 155,A -35.7861,B 21.3921,C -0.8011,E1 21.5397,E2 843.3472} C_DIS
LIN {X 112.05,Y -70.2762,Z 155,A -33.8184,B 21.3919,C -0.8079,E1 21.5427,E2 841.3727} C_DIS
LIN {X 114.3103,Y -66.5361,Z 155,A -31.9192,B 21.3917,C -0.8135,E1 21.5454,E2 839.4696} C_DIS
LIN {X 116.5937,Y -62.4479,Z 155,A -29.742,B 21.3912,C -0.8265,E1 21.5483,E2 837.2705} C_DIS
LIN {X 118.9023,Y -57.9305,Z 155,A -27.8826,B 21.3916,C -0.8168,E1 21.5506,E2 835.4493} C_DIS
LIN {X 120.117,Y -55.3643,Z 155,A -26.6121,B 21.3914,C -0.8225,E1 21.5521,E2 834.1717} C_DIS
LIN {X 121.7466,Y -51.6881,Z 155,A -24.9276,B 21.3913,C -0.8249,E1 21.554,E2 832.4915} C_DIS
LIN {X 123.4256,Y -47.5351,Z 155,A -22.9541,B 21.391,C -0.8324,E1 21.556,E2 830.5105} C_DIS
Enddeposition()
END
